// TIA Portal V17 export
// export: Created 2024-09-02T12:50:07.0584181Z, ExportSetting WithDefaults, DisplayName Totally Integrated Automation Portal, DisplayVersion V17, DisplayName TIA Portal Openness, DisplayVersion V17, DisplayName TIA Portal Version Control Interface, DisplayVersion V17, DisplayName STEP 7 Professional, DisplayVersion V17, DisplayName STEP 7 Safety, DisplayVersion V17, DisplayName WinCC Professional, DisplayVersion V17
FUNCTION "AnwFC2_FG01_Station_OP70" : Void   // FC1282, LAD
TITLE = Station
{ S7_Optimized_Access := 'TRUE' }
AUTHOR : VAF
FAMILY : SK
NAME : SK
VERSION : 0.1
// stored: AutoNumber false, IsIECCheckEnabled false, SetENOAutomatically false, UDAEnableTagReadback false
   VAR_TEMP
      Motion_Release : Bool;   // Motion permit
      Hand : Bool;
      Auto : Bool;
      t_Ret_Val_SFC : Int;
      t_fm_Gen : Bool;
      t_ParityFault : Bool;
      t_ConfigFault : Bool;
      t_Retval : Bool;
      MM90_AS : Bool;
      MM90_GS : Bool;
      X1 : Int;
      X2 : Int;
      Y : Int;
      X_actual : Int;
   END_VAR
   VAR_TEMP   // added for the SCL form of the ladder/FBD networks
      _w1 : Bool;
      _w2 : Bool;
   END_VAR
BEGIN

REGION Network 1: Motion permit / Hand/ Auto
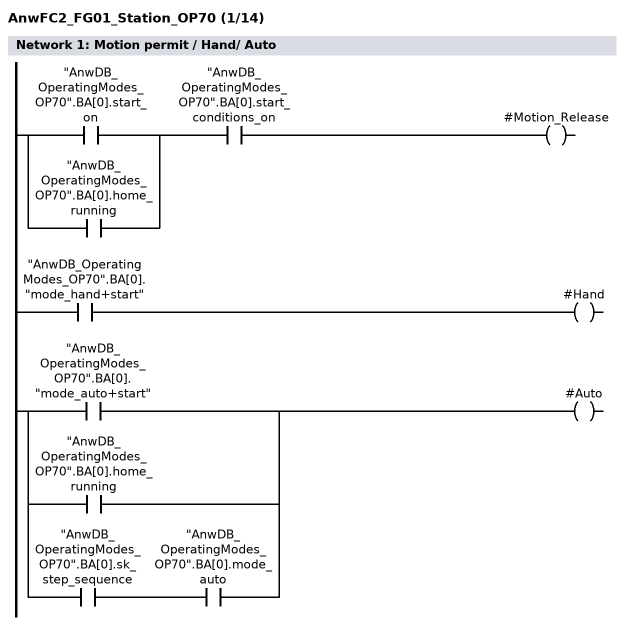
   RUNG wire#powerrail
      Contact( "AnwDB_OperatingModes_OP70".BA[0].start_on )
      wire#w1
      Contact( "AnwDB_OperatingModes_OP70".BA[0].start_conditions_on )
      Coil( #Motion_Release )
   END_RUNG
   RUNG wire#powerrail
      Contact( "AnwDB_OperatingModes_OP70".BA[0].home_running )
   END_RUNG wire#w1
   RUNG wire#powerrail
      Contact( "AnwDB_OperatingModes_OP70".BA[0]."mode_hand+start" )
      Coil( #Hand )
   END_RUNG
   RUNG wire#powerrail
      Contact( "AnwDB_OperatingModes_OP70".BA[0]."mode_auto+start" )
      wire#w2
      Coil( #Auto )
   END_RUNG
   RUNG wire#powerrail
      Contact( "AnwDB_OperatingModes_OP70".BA[0].home_running )
   END_RUNG wire#w2
   RUNG wire#powerrail
      Contact( "AnwDB_OperatingModes_OP70".BA[0].sk_step_sequence )
      Contact( "AnwDB_OperatingModes_OP70".BA[0].mode_auto )
   END_RUNG wire#w2
   // the same network as SCL:
   #Motion_Release := ("AnwDB_OperatingModes_OP70".BA[0].start_on OR "AnwDB_OperatingModes_OP70".BA[0].home_running) AND "AnwDB_OperatingModes_OP70".BA[0].start_conditions_on;
   #Hand := "AnwDB_OperatingModes_OP70".BA[0]."mode_hand+start";
   #Auto := "AnwDB_OperatingModes_OP70".BA[0]."mode_auto+start" OR "AnwDB_OperatingModes_OP70".BA[0].home_running OR ("AnwDB_OperatingModes_OP70".BA[0].sk_step_sequence AND "AnwDB_OperatingModes_OP70".BA[0].mode_auto);
END_REGION

REGION Network 2: Call of the step sequence
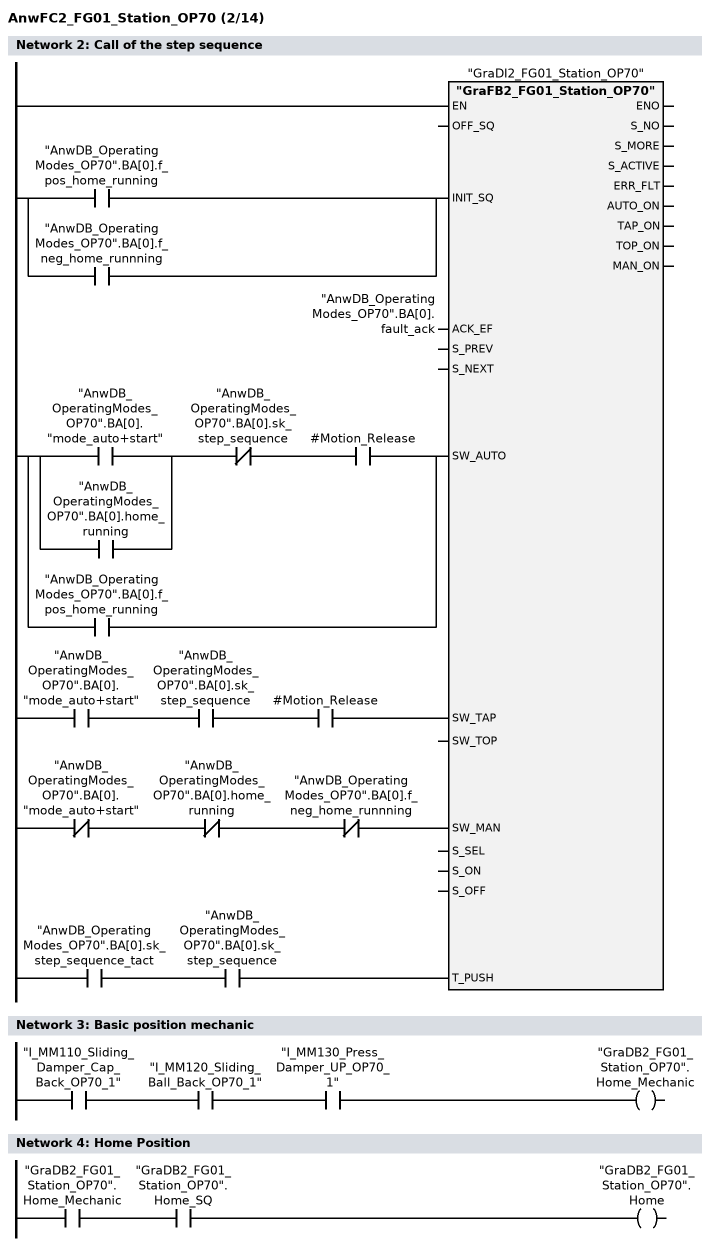
   RUNG wire#powerrail
      "GraDI2_FG01_Station_OP70"(INIT_SQ := wire#w1, SW_AUTO := wire#w3, SW_TAP := wire#w4, SW_MAN := wire#w5, T_PUSH := wire#w6, OFF_SQ :=, ACK_EF := "AnwDB_OperatingModes_OP70".BA[0].fault_ack, S_PREV :=, S_NEXT :=, SW_TOP :=, S_SEL :=, S_ON :=, S_OFF :=, S_NO =>, S_MORE =>, S_ACTIVE =>, ERR_FLT =>, AUTO_ON =>, TAP_ON =>, TOP_ON =>, MAN_ON =>)
   END_RUNG
   RUNG wire#powerrail
      Contact( "AnwDB_OperatingModes_OP70".BA[0].f_pos_home_running )
   END_RUNG wire#w1
   RUNG wire#powerrail
      Contact( "AnwDB_OperatingModes_OP70".BA[0].f_neg_home_runnning )
   END_RUNG wire#w1
   RUNG wire#powerrail
      Contact( "AnwDB_OperatingModes_OP70".BA[0]."mode_auto+start" )
      wire#w2
      I_Contact( "AnwDB_OperatingModes_OP70".BA[0].sk_step_sequence )
      Contact( #Motion_Release )
   END_RUNG wire#w3
   RUNG wire#powerrail
      Contact( "AnwDB_OperatingModes_OP70".BA[0].home_running )
   END_RUNG wire#w2
   RUNG wire#powerrail
      Contact( "AnwDB_OperatingModes_OP70".BA[0].f_pos_home_running )
   END_RUNG wire#w3
   RUNG wire#powerrail
      Contact( "AnwDB_OperatingModes_OP70".BA[0]."mode_auto+start" )
      Contact( "AnwDB_OperatingModes_OP70".BA[0].sk_step_sequence )
      Contact( #Motion_Release )
   END_RUNG wire#w4
   RUNG wire#powerrail
      I_Contact( "AnwDB_OperatingModes_OP70".BA[0]."mode_auto+start" )
      I_Contact( "AnwDB_OperatingModes_OP70".BA[0].home_running )
      I_Contact( "AnwDB_OperatingModes_OP70".BA[0].f_neg_home_runnning )
   END_RUNG wire#w5
   RUNG wire#powerrail
      Contact( "AnwDB_OperatingModes_OP70".BA[0].sk_step_sequence_tact )
      Contact( "AnwDB_OperatingModes_OP70".BA[0].sk_step_sequence )
   END_RUNG wire#w6
   // the same network as SCL:
   "GraDI2_FG01_Station_OP70"(INIT_SQ := "AnwDB_OperatingModes_OP70".BA[0].f_pos_home_running OR "AnwDB_OperatingModes_OP70".BA[0].f_neg_home_runnning,   // "GraFB2_FG01_Station_OP70"
                           ACK_EF := "AnwDB_OperatingModes_OP70".BA[0].fault_ack,
                           SW_AUTO := (("AnwDB_OperatingModes_OP70".BA[0]."mode_auto+start" OR "AnwDB_OperatingModes_OP70".BA[0].home_running) AND NOT "AnwDB_OperatingModes_OP70".BA[0].sk_step_sequence AND #Motion_Release) OR "AnwDB_OperatingModes_OP70".BA[0].f_pos_home_running,
                           SW_TAP := "AnwDB_OperatingModes_OP70".BA[0]."mode_auto+start" AND "AnwDB_OperatingModes_OP70".BA[0].sk_step_sequence AND #Motion_Release,
                           SW_MAN := NOT "AnwDB_OperatingModes_OP70".BA[0]."mode_auto+start" AND NOT "AnwDB_OperatingModes_OP70".BA[0].home_running AND NOT "AnwDB_OperatingModes_OP70".BA[0].f_neg_home_runnning,
                           T_PUSH := "AnwDB_OperatingModes_OP70".BA[0].sk_step_sequence_tact AND "AnwDB_OperatingModes_OP70".BA[0].sk_step_sequence);
END_REGION

REGION Network 3: Basic position mechanic
   RUNG wire#powerrail
      Contact( "I_MM110_Sliding_Damper_Cap_Back_OP70_1" )
      Contact( "I_MM120_Sliding_Ball_Back_OP70_1" )
      Contact( "I_MM130_Press_Damper_UP_OP70_1" )
      Coil( "GraDB2_FG01_Station_OP70".Home_Mechanic )
   END_RUNG
   // the same network as SCL:
   "GraDB2_FG01_Station_OP70".Home_Mechanic := "I_MM110_Sliding_Damper_Cap_Back_OP70_1" AND "I_MM120_Sliding_Ball_Back_OP70_1" AND "I_MM130_Press_Damper_UP_OP70_1";
END_REGION

REGION Network 4: Home Position
   RUNG wire#powerrail
      Contact( "GraDB2_FG01_Station_OP70".Home_Mechanic )
      Contact( "GraDB2_FG01_Station_OP70".Home_SQ )
      Coil( "GraDB2_FG01_Station_OP70".Home )
   END_RUNG
   // the same network as SCL:
   "GraDB2_FG01_Station_OP70".Home := "GraDB2_FG01_Station_OP70".Home_Mechanic AND "GraDB2_FG01_Station_OP70".Home_SQ;
END_REGION

REGION Network 5: ########### USER ###########
END_REGION

REGION Network 6: Screen selection with NOK BEA1
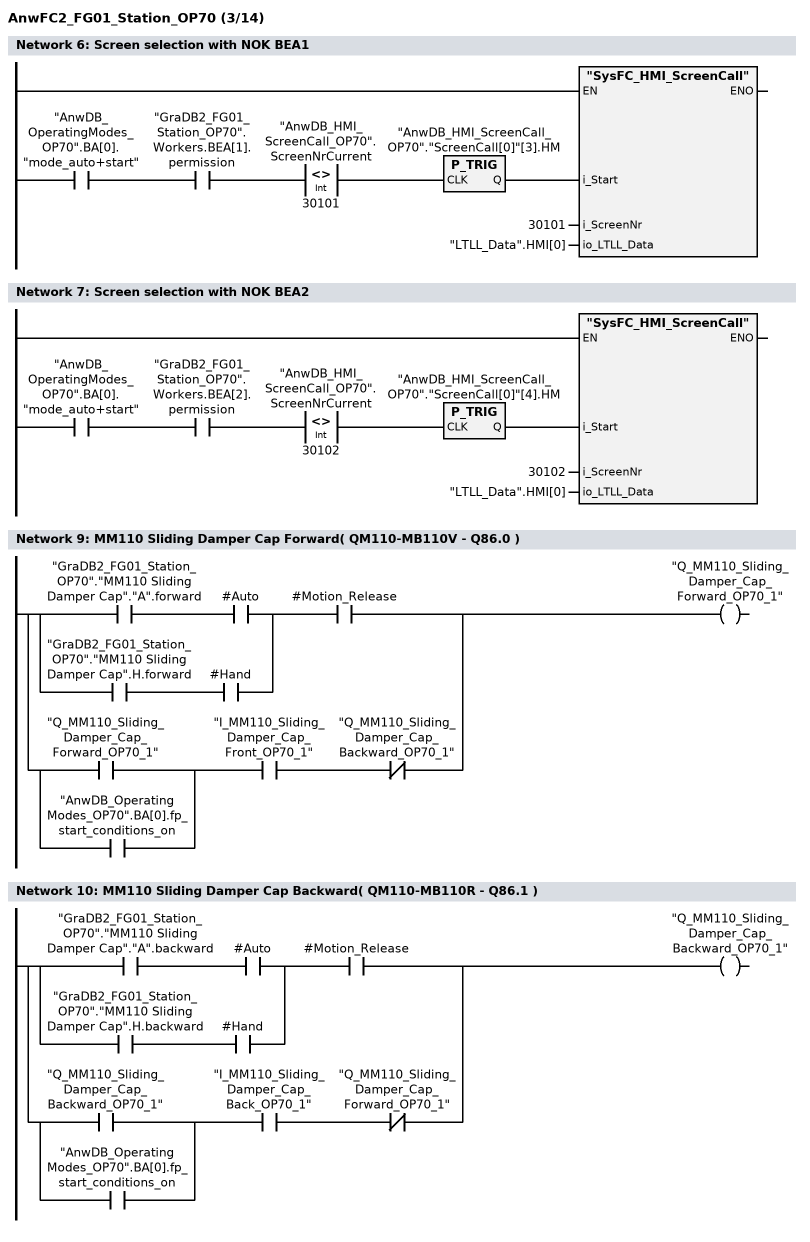
   RUNG wire#powerrail
      "SysFC_HMI_ScreenCall"(i_Start := wire#w1, i_ScreenNr := 30101, io_LTLL_Data := "LTLL_Data".HMI[0])
   END_RUNG
   RUNG wire#powerrail
      Contact( "AnwDB_OperatingModes_OP70".BA[0]."mode_auto+start" )
      Contact( "GraDB2_FG01_Station_OP70".Workers.BEA[1].permission )
      { S7_Templates := "SrcType := Int" } NE_Contact(in1 := "AnwDB_HMI_ScreenCall_OP70".ScreenNrCurrent, in2 := 30101)
      P_Trig( "AnwDB_HMI_ScreenCall_OP70"."ScreenCall[0]"[3].HM )
   END_RUNG wire#w1
   // the same network as SCL:
   #_w1 := "AnwDB_OperatingModes_OP70".BA[0]."mode_auto+start" AND "GraDB2_FG01_Station_OP70".Workers.BEA[1].permission AND ("AnwDB_HMI_ScreenCall_OP70".ScreenNrCurrent <> 30101);
   #_w2 := #_w1 AND NOT "AnwDB_HMI_ScreenCall_OP70"."ScreenCall[0]"[3].HM;   // rising edge
   "AnwDB_HMI_ScreenCall_OP70"."ScreenCall[0]"[3].HM := #_w1;
   "SysFC_HMI_ScreenCall"(i_Start := #_w2, i_ScreenNr := 30101, io_LTLL_Data := "LTLL_Data".HMI[0]);
END_REGION

REGION Network 7: Screen selection with NOK BEA2
   RUNG wire#powerrail
      "SysFC_HMI_ScreenCall"(i_Start := wire#w1, i_ScreenNr := 30102, io_LTLL_Data := "LTLL_Data".HMI[0])
   END_RUNG
   RUNG wire#powerrail
      Contact( "AnwDB_OperatingModes_OP70".BA[0]."mode_auto+start" )
      Contact( "GraDB2_FG01_Station_OP70".Workers.BEA[2].permission )
      { S7_Templates := "SrcType := Int" } NE_Contact(in1 := "AnwDB_HMI_ScreenCall_OP70".ScreenNrCurrent, in2 := 30102)
      P_Trig( "AnwDB_HMI_ScreenCall_OP70"."ScreenCall[0]"[4].HM )
   END_RUNG wire#w1
   // the same network as SCL:
   #_w1 := "AnwDB_OperatingModes_OP70".BA[0]."mode_auto+start" AND "GraDB2_FG01_Station_OP70".Workers.BEA[2].permission AND ("AnwDB_HMI_ScreenCall_OP70".ScreenNrCurrent <> 30102);
   #_w2 := #_w1 AND NOT "AnwDB_HMI_ScreenCall_OP70"."ScreenCall[0]"[4].HM;   // rising edge
   "AnwDB_HMI_ScreenCall_OP70"."ScreenCall[0]"[4].HM := #_w1;
   "SysFC_HMI_ScreenCall"(i_Start := #_w2, i_ScreenNr := 30102, io_LTLL_Data := "LTLL_Data".HMI[0]);
END_REGION

REGION Network 8: ########### SS_02_001_Setup ###########
END_REGION

REGION Network 9: MM110 Sliding Damper Cap Forward( QM110-MB110V - Q86.0 )
   RUNG wire#powerrail
      Contact( "GraDB2_FG01_Station_OP70"."MM110 Sliding Damper Cap"."A".forward )
      Contact( #Auto )
      wire#w1
      Contact( #Motion_Release )
      wire#w2
      Coil( "Q_MM110_Sliding_Damper_Cap_Forward_OP70_1" )
   END_RUNG
   RUNG wire#powerrail
      Contact( "GraDB2_FG01_Station_OP70"."MM110 Sliding Damper Cap".H.forward )
      Contact( #Hand )
   END_RUNG wire#w1
   RUNG wire#powerrail
      Contact( "Q_MM110_Sliding_Damper_Cap_Forward_OP70_1" )
      wire#w3
      Contact( "I_MM110_Sliding_Damper_Cap_Front_OP70_1" )
      I_Contact( "Q_MM110_Sliding_Damper_Cap_Backward_OP70_1" )
   END_RUNG wire#w2
   RUNG wire#powerrail
      Contact( "AnwDB_OperatingModes_OP70".BA[0].fp_start_conditions_on )
   END_RUNG wire#w3
   // the same network as SCL:
   "Q_MM110_Sliding_Damper_Cap_Forward_OP70_1" := ((("GraDB2_FG01_Station_OP70"."MM110 Sliding Damper Cap"."A".forward AND #Auto) OR ("GraDB2_FG01_Station_OP70"."MM110 Sliding Damper Cap".H.forward AND #Hand)) AND #Motion_Release) OR (("Q_MM110_Sliding_Damper_Cap_Forward_OP70_1" OR "AnwDB_OperatingModes_OP70".BA[0].fp_start_conditions_on) AND "I_MM110_Sliding_Damper_Cap_Front_OP70_1" AND NOT "Q_MM110_Sliding_Damper_Cap_Backward_OP70_1");
END_REGION

REGION Network 10: MM110 Sliding Damper Cap Backward( QM110-MB110R - Q86.1 )
   RUNG wire#powerrail
      Contact( "GraDB2_FG01_Station_OP70"."MM110 Sliding Damper Cap"."A".backward )
      Contact( #Auto )
      wire#w1
      Contact( #Motion_Release )
      wire#w2
      Coil( "Q_MM110_Sliding_Damper_Cap_Backward_OP70_1" )
   END_RUNG
   RUNG wire#powerrail
      Contact( "GraDB2_FG01_Station_OP70"."MM110 Sliding Damper Cap".H.backward )
      Contact( #Hand )
   END_RUNG wire#w1
   RUNG wire#powerrail
      Contact( "Q_MM110_Sliding_Damper_Cap_Backward_OP70_1" )
      wire#w3
      Contact( "I_MM110_Sliding_Damper_Cap_Back_OP70_1" )
      I_Contact( "Q_MM110_Sliding_Damper_Cap_Forward_OP70_1" )
   END_RUNG wire#w2
   RUNG wire#powerrail
      Contact( "AnwDB_OperatingModes_OP70".BA[0].fp_start_conditions_on )
   END_RUNG wire#w3
   // the same network as SCL:
   "Q_MM110_Sliding_Damper_Cap_Backward_OP70_1" := ((("GraDB2_FG01_Station_OP70"."MM110 Sliding Damper Cap"."A".backward AND #Auto) OR ("GraDB2_FG01_Station_OP70"."MM110 Sliding Damper Cap".H.backward AND #Hand)) AND #Motion_Release) OR (("Q_MM110_Sliding_Damper_Cap_Backward_OP70_1" OR "AnwDB_OperatingModes_OP70".BA[0].fp_start_conditions_on) AND "I_MM110_Sliding_Damper_Cap_Back_OP70_1" AND NOT "Q_MM110_Sliding_Damper_Cap_Forward_OP70_1");
END_REGION

REGION Network 11: Hand line(13)
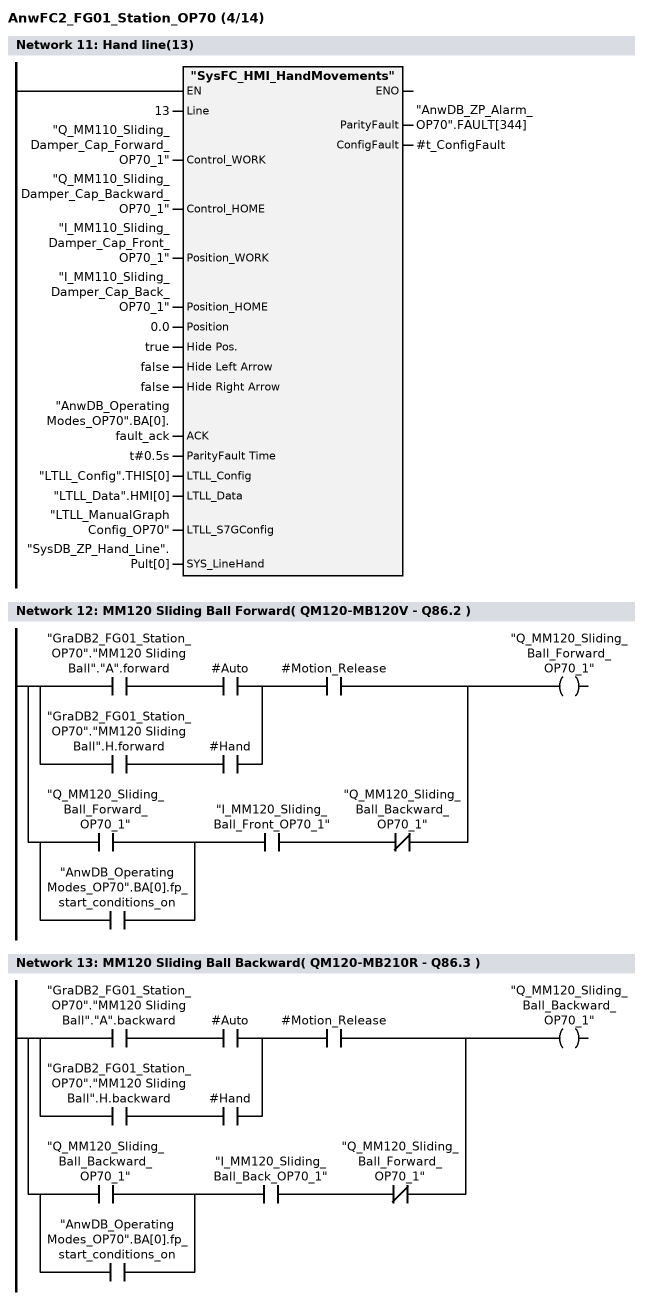
   RUNG wire#powerrail
      "SysFC_HMI_HandMovements"(Line := 13, Control_WORK := "Q_MM110_Sliding_Damper_Cap_Forward_OP70_1", Control_HOME := "Q_MM110_Sliding_Damper_Cap_Backward_OP70_1", Position_WORK := "I_MM110_Sliding_Damper_Cap_Front_OP70_1", Position_HOME := "I_MM110_Sliding_Damper_Cap_Back_OP70_1", Position := 0.0, "Hide Pos." := true, "Hide Left Arrow" := false, "Hide Right Arrow" := false, ACK := "AnwDB_OperatingModes_OP70".BA[0].fault_ack, "ParityFault Time" := t#0.5s, LTLL_Config := "LTLL_Config".THIS[0], LTLL_Data := "LTLL_Data".HMI[0], LTLL_S7GConfig := "LTLL_ManualGraphConfig_OP70", SYS_LineHand := "SysDB_ZP_Hand_Line".Pult[0], ParityFault => "AnwDB_ZP_Alarm_OP70".FAULT[344], ConfigFault => #t_ConfigFault)
   END_RUNG
   // the same network as SCL:
   "SysFC_HMI_HandMovements"(Line := 13,
                           Control_WORK := "Q_MM110_Sliding_Damper_Cap_Forward_OP70_1",
                           Control_HOME := "Q_MM110_Sliding_Damper_Cap_Backward_OP70_1",
                           Position_WORK := "I_MM110_Sliding_Damper_Cap_Front_OP70_1",
                           Position_HOME := "I_MM110_Sliding_Damper_Cap_Back_OP70_1",
                           Position := 0.0,
                           "Hide Pos." := true,
                           "Hide Left Arrow" := false,
                           "Hide Right Arrow" := false,
                           ACK := "AnwDB_OperatingModes_OP70".BA[0].fault_ack,
                           "ParityFault Time" := t#0.5s,
                           LTLL_Config := "LTLL_Config".THIS[0],
                           LTLL_Data := "LTLL_Data".HMI[0],
                           LTLL_S7GConfig := "LTLL_ManualGraphConfig_OP70",
                           SYS_LineHand := "SysDB_ZP_Hand_Line".Pult[0],
                           ParityFault => "AnwDB_ZP_Alarm_OP70".FAULT[344],
                           ConfigFault => #t_ConfigFault);
END_REGION

REGION Network 12: MM120 Sliding Ball Forward( QM120-MB120V - Q86.2 )
   RUNG wire#powerrail
      Contact( "GraDB2_FG01_Station_OP70"."MM120 Sliding Ball"."A".forward )
      Contact( #Auto )
      wire#w1
      Contact( #Motion_Release )
      wire#w2
      Coil( "Q_MM120_Sliding_Ball_Forward_OP70_1" )
   END_RUNG
   RUNG wire#powerrail
      Contact( "GraDB2_FG01_Station_OP70"."MM120 Sliding Ball".H.forward )
      Contact( #Hand )
   END_RUNG wire#w1
   RUNG wire#powerrail
      Contact( "Q_MM120_Sliding_Ball_Forward_OP70_1" )
      wire#w3
      Contact( "I_MM120_Sliding_Ball_Front_OP70_1" )
      I_Contact( "Q_MM120_Sliding_Ball_Backward_OP70_1" )
   END_RUNG wire#w2
   RUNG wire#powerrail
      Contact( "AnwDB_OperatingModes_OP70".BA[0].fp_start_conditions_on )
   END_RUNG wire#w3
   // the same network as SCL:
   "Q_MM120_Sliding_Ball_Forward_OP70_1" := ((("GraDB2_FG01_Station_OP70"."MM120 Sliding Ball"."A".forward AND #Auto) OR ("GraDB2_FG01_Station_OP70"."MM120 Sliding Ball".H.forward AND #Hand)) AND #Motion_Release) OR (("Q_MM120_Sliding_Ball_Forward_OP70_1" OR "AnwDB_OperatingModes_OP70".BA[0].fp_start_conditions_on) AND "I_MM120_Sliding_Ball_Front_OP70_1" AND NOT "Q_MM120_Sliding_Ball_Backward_OP70_1");
END_REGION

REGION Network 13: MM120 Sliding Ball Backward( QM120-MB210R - Q86.3 )
   RUNG wire#powerrail
      Contact( "GraDB2_FG01_Station_OP70"."MM120 Sliding Ball"."A".backward )
      Contact( #Auto )
      wire#w1
      Contact( #Motion_Release )
      wire#w2
      Coil( "Q_MM120_Sliding_Ball_Backward_OP70_1" )
   END_RUNG
   RUNG wire#powerrail
      Contact( "GraDB2_FG01_Station_OP70"."MM120 Sliding Ball".H.backward )
      Contact( #Hand )
   END_RUNG wire#w1
   RUNG wire#powerrail
      Contact( "Q_MM120_Sliding_Ball_Backward_OP70_1" )
      wire#w3
      Contact( "I_MM120_Sliding_Ball_Back_OP70_1" )
      I_Contact( "Q_MM120_Sliding_Ball_Forward_OP70_1" )
   END_RUNG wire#w2
   RUNG wire#powerrail
      Contact( "AnwDB_OperatingModes_OP70".BA[0].fp_start_conditions_on )
   END_RUNG wire#w3
   // the same network as SCL:
   "Q_MM120_Sliding_Ball_Backward_OP70_1" := ((("GraDB2_FG01_Station_OP70"."MM120 Sliding Ball"."A".backward AND #Auto) OR ("GraDB2_FG01_Station_OP70"."MM120 Sliding Ball".H.backward AND #Hand)) AND #Motion_Release) OR (("Q_MM120_Sliding_Ball_Backward_OP70_1" OR "AnwDB_OperatingModes_OP70".BA[0].fp_start_conditions_on) AND "I_MM120_Sliding_Ball_Back_OP70_1" AND NOT "Q_MM120_Sliding_Ball_Forward_OP70_1");
END_REGION

REGION Network 14: Hand line(14)
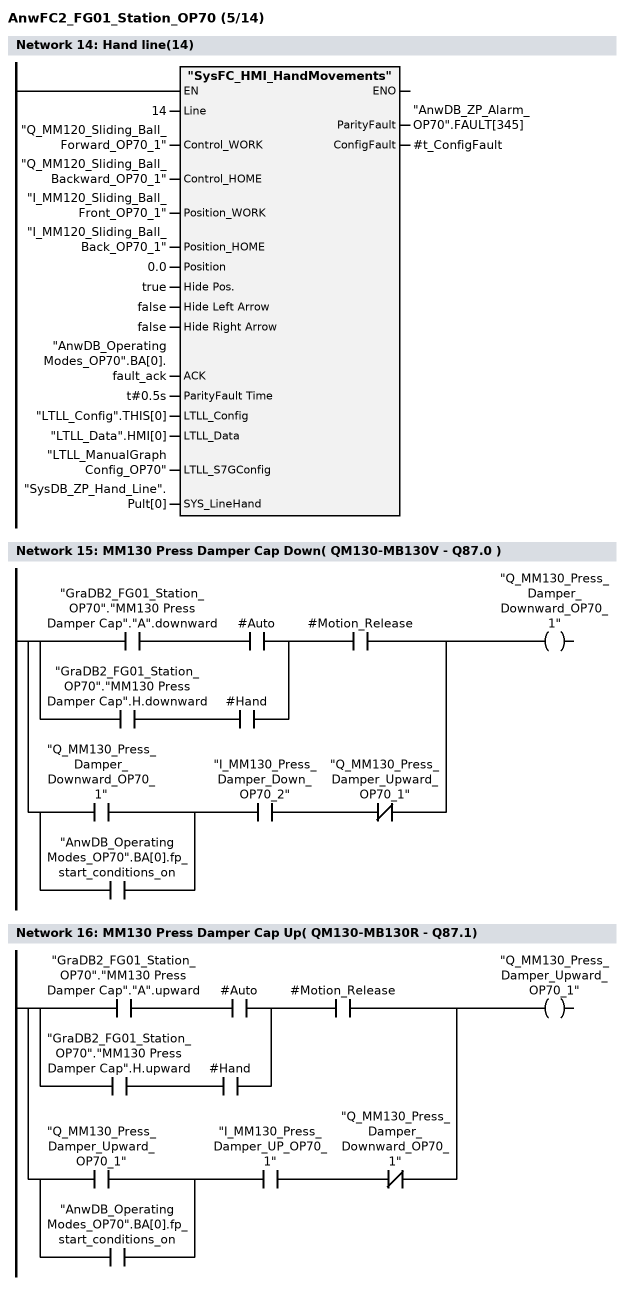
   RUNG wire#powerrail
      "SysFC_HMI_HandMovements"(Line := 14, Control_WORK := "Q_MM120_Sliding_Ball_Forward_OP70_1", Control_HOME := "Q_MM120_Sliding_Ball_Backward_OP70_1", Position_WORK := "I_MM120_Sliding_Ball_Front_OP70_1", Position_HOME := "I_MM120_Sliding_Ball_Back_OP70_1", Position := 0.0, "Hide Pos." := true, "Hide Left Arrow" := false, "Hide Right Arrow" := false, ACK := "AnwDB_OperatingModes_OP70".BA[0].fault_ack, "ParityFault Time" := t#0.5s, LTLL_Config := "LTLL_Config".THIS[0], LTLL_Data := "LTLL_Data".HMI[0], LTLL_S7GConfig := "LTLL_ManualGraphConfig_OP70", SYS_LineHand := "SysDB_ZP_Hand_Line".Pult[0], ParityFault => "AnwDB_ZP_Alarm_OP70".FAULT[345], ConfigFault => #t_ConfigFault)
   END_RUNG
   // the same network as SCL:
   "SysFC_HMI_HandMovements"(Line := 14,
                           Control_WORK := "Q_MM120_Sliding_Ball_Forward_OP70_1",
                           Control_HOME := "Q_MM120_Sliding_Ball_Backward_OP70_1",
                           Position_WORK := "I_MM120_Sliding_Ball_Front_OP70_1",
                           Position_HOME := "I_MM120_Sliding_Ball_Back_OP70_1",
                           Position := 0.0,
                           "Hide Pos." := true,
                           "Hide Left Arrow" := false,
                           "Hide Right Arrow" := false,
                           ACK := "AnwDB_OperatingModes_OP70".BA[0].fault_ack,
                           "ParityFault Time" := t#0.5s,
                           LTLL_Config := "LTLL_Config".THIS[0],
                           LTLL_Data := "LTLL_Data".HMI[0],
                           LTLL_S7GConfig := "LTLL_ManualGraphConfig_OP70",
                           SYS_LineHand := "SysDB_ZP_Hand_Line".Pult[0],
                           ParityFault => "AnwDB_ZP_Alarm_OP70".FAULT[345],
                           ConfigFault => #t_ConfigFault);
END_REGION

REGION Network 15: MM130 Press Damper Cap Down( QM130-MB130V - Q87.0 )
   RUNG wire#powerrail
      Contact( "GraDB2_FG01_Station_OP70"."MM130 Press Damper Cap"."A".downward )
      Contact( #Auto )
      wire#w1
      Contact( #Motion_Release )
      wire#w2
      Coil( "Q_MM130_Press_Damper_Downward_OP70_1" )
   END_RUNG
   RUNG wire#powerrail
      Contact( "GraDB2_FG01_Station_OP70"."MM130 Press Damper Cap".H.downward )
      Contact( #Hand )
   END_RUNG wire#w1
   RUNG wire#powerrail
      Contact( "Q_MM130_Press_Damper_Downward_OP70_1" )
      wire#w3
      Contact( "I_MM130_Press_Damper_Down_OP70_2" )
      I_Contact( "Q_MM130_Press_Damper_Upward_OP70_1" )
   END_RUNG wire#w2
   RUNG wire#powerrail
      Contact( "AnwDB_OperatingModes_OP70".BA[0].fp_start_conditions_on )
   END_RUNG wire#w3
   // the same network as SCL:
   "Q_MM130_Press_Damper_Downward_OP70_1" := ((("GraDB2_FG01_Station_OP70"."MM130 Press Damper Cap"."A".downward AND #Auto) OR ("GraDB2_FG01_Station_OP70"."MM130 Press Damper Cap".H.downward AND #Hand)) AND #Motion_Release) OR (("Q_MM130_Press_Damper_Downward_OP70_1" OR "AnwDB_OperatingModes_OP70".BA[0].fp_start_conditions_on) AND "I_MM130_Press_Damper_Down_OP70_2" AND NOT "Q_MM130_Press_Damper_Upward_OP70_1");
END_REGION

REGION Network 16: MM130 Press Damper Cap Up( QM130-MB130R - Q87.1)
   RUNG wire#powerrail
      Contact( "GraDB2_FG01_Station_OP70"."MM130 Press Damper Cap"."A".upward )
      Contact( #Auto )
      wire#w1
      Contact( #Motion_Release )
      wire#w2
      Coil( "Q_MM130_Press_Damper_Upward_OP70_1" )
   END_RUNG
   RUNG wire#powerrail
      Contact( "GraDB2_FG01_Station_OP70"."MM130 Press Damper Cap".H.upward )
      Contact( #Hand )
   END_RUNG wire#w1
   RUNG wire#powerrail
      Contact( "Q_MM130_Press_Damper_Upward_OP70_1" )
      wire#w3
      Contact( "I_MM130_Press_Damper_UP_OP70_1" )
      I_Contact( "Q_MM130_Press_Damper_Downward_OP70_1" )
   END_RUNG wire#w2
   RUNG wire#powerrail
      Contact( "AnwDB_OperatingModes_OP70".BA[0].fp_start_conditions_on )
   END_RUNG wire#w3
   // the same network as SCL:
   "Q_MM130_Press_Damper_Upward_OP70_1" := ((("GraDB2_FG01_Station_OP70"."MM130 Press Damper Cap"."A".upward AND #Auto) OR ("GraDB2_FG01_Station_OP70"."MM130 Press Damper Cap".H.upward AND #Hand)) AND #Motion_Release) OR (("Q_MM130_Press_Damper_Upward_OP70_1" OR "AnwDB_OperatingModes_OP70".BA[0].fp_start_conditions_on) AND "I_MM130_Press_Damper_UP_OP70_1" AND NOT "Q_MM130_Press_Damper_Downward_OP70_1");
END_REGION

REGION Network 17: Hand line(15)
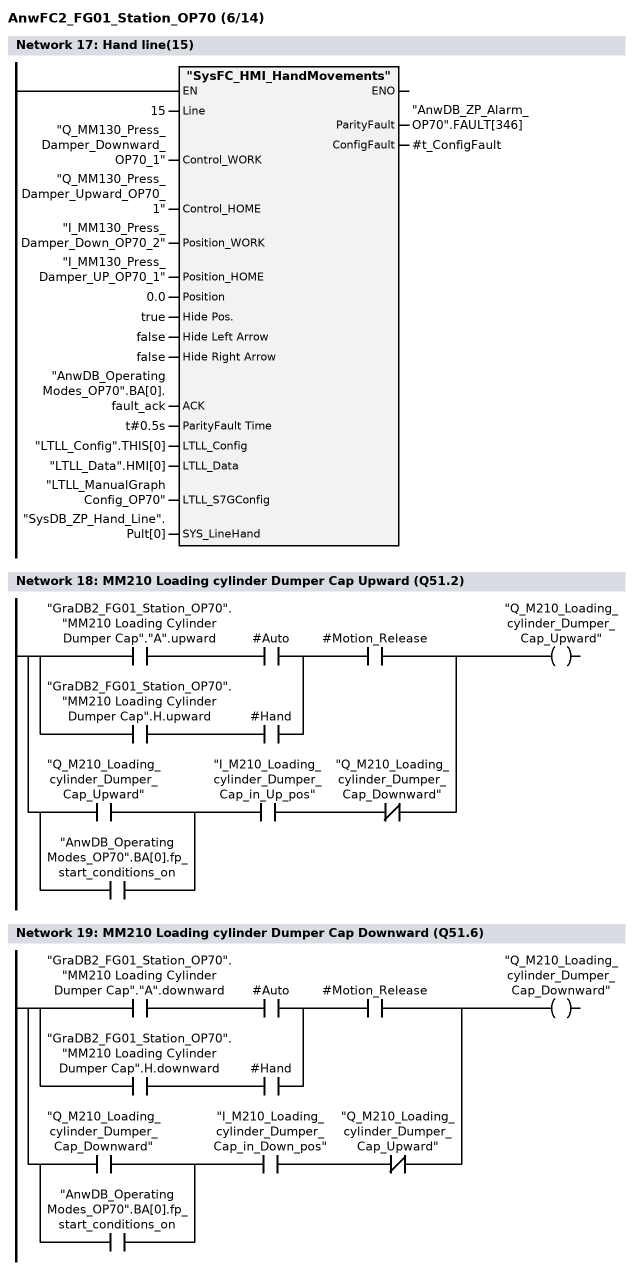
   RUNG wire#powerrail
      "SysFC_HMI_HandMovements"(Line := 15, Control_WORK := "Q_MM130_Press_Damper_Downward_OP70_1", Control_HOME := "Q_MM130_Press_Damper_Upward_OP70_1", Position_WORK := "I_MM130_Press_Damper_Down_OP70_2", Position_HOME := "I_MM130_Press_Damper_UP_OP70_1", Position := 0.0, "Hide Pos." := true, "Hide Left Arrow" := false, "Hide Right Arrow" := false, ACK := "AnwDB_OperatingModes_OP70".BA[0].fault_ack, "ParityFault Time" := t#0.5s, LTLL_Config := "LTLL_Config".THIS[0], LTLL_Data := "LTLL_Data".HMI[0], LTLL_S7GConfig := "LTLL_ManualGraphConfig_OP70", SYS_LineHand := "SysDB_ZP_Hand_Line".Pult[0], ParityFault => "AnwDB_ZP_Alarm_OP70".FAULT[346], ConfigFault => #t_ConfigFault)
   END_RUNG
   // the same network as SCL:
   "SysFC_HMI_HandMovements"(Line := 15,
                           Control_WORK := "Q_MM130_Press_Damper_Downward_OP70_1",
                           Control_HOME := "Q_MM130_Press_Damper_Upward_OP70_1",
                           Position_WORK := "I_MM130_Press_Damper_Down_OP70_2",
                           Position_HOME := "I_MM130_Press_Damper_UP_OP70_1",
                           Position := 0.0,
                           "Hide Pos." := true,
                           "Hide Left Arrow" := false,
                           "Hide Right Arrow" := false,
                           ACK := "AnwDB_OperatingModes_OP70".BA[0].fault_ack,
                           "ParityFault Time" := t#0.5s,
                           LTLL_Config := "LTLL_Config".THIS[0],
                           LTLL_Data := "LTLL_Data".HMI[0],
                           LTLL_S7GConfig := "LTLL_ManualGraphConfig_OP70",
                           SYS_LineHand := "SysDB_ZP_Hand_Line".Pult[0],
                           ParityFault => "AnwDB_ZP_Alarm_OP70".FAULT[346],
                           ConfigFault => #t_ConfigFault);
END_REGION

REGION Network 18: MM210 Loading cylinder Dumper Cap Upward (Q51.2)
   RUNG wire#powerrail
      Contact( "GraDB2_FG01_Station_OP70"."MM210 Loading Cylinder Dumper Cap"."A".upward )
      Contact( #Auto )
      wire#w1
      Contact( #Motion_Release )
      wire#w2
      Coil( "Q_M210_Loading_cylinder_Dumper_Cap_Upward" )
   END_RUNG
   RUNG wire#powerrail
      Contact( "GraDB2_FG01_Station_OP70"."MM210 Loading Cylinder Dumper Cap".H.upward )
      Contact( #Hand )
   END_RUNG wire#w1
   RUNG wire#powerrail
      Contact( "Q_M210_Loading_cylinder_Dumper_Cap_Upward" )
      wire#w3
      Contact( "I_M210_Loading_cylinder_Dumper_Cap_in_Up_pos" )
      I_Contact( "Q_M210_Loading_cylinder_Dumper_Cap_Downward" )
   END_RUNG wire#w2
   RUNG wire#powerrail
      Contact( "AnwDB_OperatingModes_OP70".BA[0].fp_start_conditions_on )
   END_RUNG wire#w3
   // the same network as SCL:
   "Q_M210_Loading_cylinder_Dumper_Cap_Upward" := ((("GraDB2_FG01_Station_OP70"."MM210 Loading Cylinder Dumper Cap"."A".upward AND #Auto) OR ("GraDB2_FG01_Station_OP70"."MM210 Loading Cylinder Dumper Cap".H.upward AND #Hand)) AND #Motion_Release) OR (("Q_M210_Loading_cylinder_Dumper_Cap_Upward" OR "AnwDB_OperatingModes_OP70".BA[0].fp_start_conditions_on) AND "I_M210_Loading_cylinder_Dumper_Cap_in_Up_pos" AND NOT "Q_M210_Loading_cylinder_Dumper_Cap_Downward");
END_REGION

REGION Network 19: MM210 Loading cylinder Dumper Cap Downward (Q51.6)
   RUNG wire#powerrail
      Contact( "GraDB2_FG01_Station_OP70"."MM210 Loading Cylinder Dumper Cap"."A".downward )
      Contact( #Auto )
      wire#w1
      Contact( #Motion_Release )
      wire#w2
      Coil( "Q_M210_Loading_cylinder_Dumper_Cap_Downward" )
   END_RUNG
   RUNG wire#powerrail
      Contact( "GraDB2_FG01_Station_OP70"."MM210 Loading Cylinder Dumper Cap".H.downward )
      Contact( #Hand )
   END_RUNG wire#w1
   RUNG wire#powerrail
      Contact( "Q_M210_Loading_cylinder_Dumper_Cap_Downward" )
      wire#w3
      Contact( "I_M210_Loading_cylinder_Dumper_Cap_in_Down_pos" )
      I_Contact( "Q_M210_Loading_cylinder_Dumper_Cap_Upward" )
   END_RUNG wire#w2
   RUNG wire#powerrail
      Contact( "AnwDB_OperatingModes_OP70".BA[0].fp_start_conditions_on )
   END_RUNG wire#w3
   // the same network as SCL:
   "Q_M210_Loading_cylinder_Dumper_Cap_Downward" := ((("GraDB2_FG01_Station_OP70"."MM210 Loading Cylinder Dumper Cap"."A".downward AND #Auto) OR ("GraDB2_FG01_Station_OP70"."MM210 Loading Cylinder Dumper Cap".H.downward AND #Hand)) AND #Motion_Release) OR (("Q_M210_Loading_cylinder_Dumper_Cap_Downward" OR "AnwDB_OperatingModes_OP70".BA[0].fp_start_conditions_on) AND "I_M210_Loading_cylinder_Dumper_Cap_in_Down_pos" AND NOT "Q_M210_Loading_cylinder_Dumper_Cap_Upward");
END_REGION

REGION Network 20: Hand linie (16)
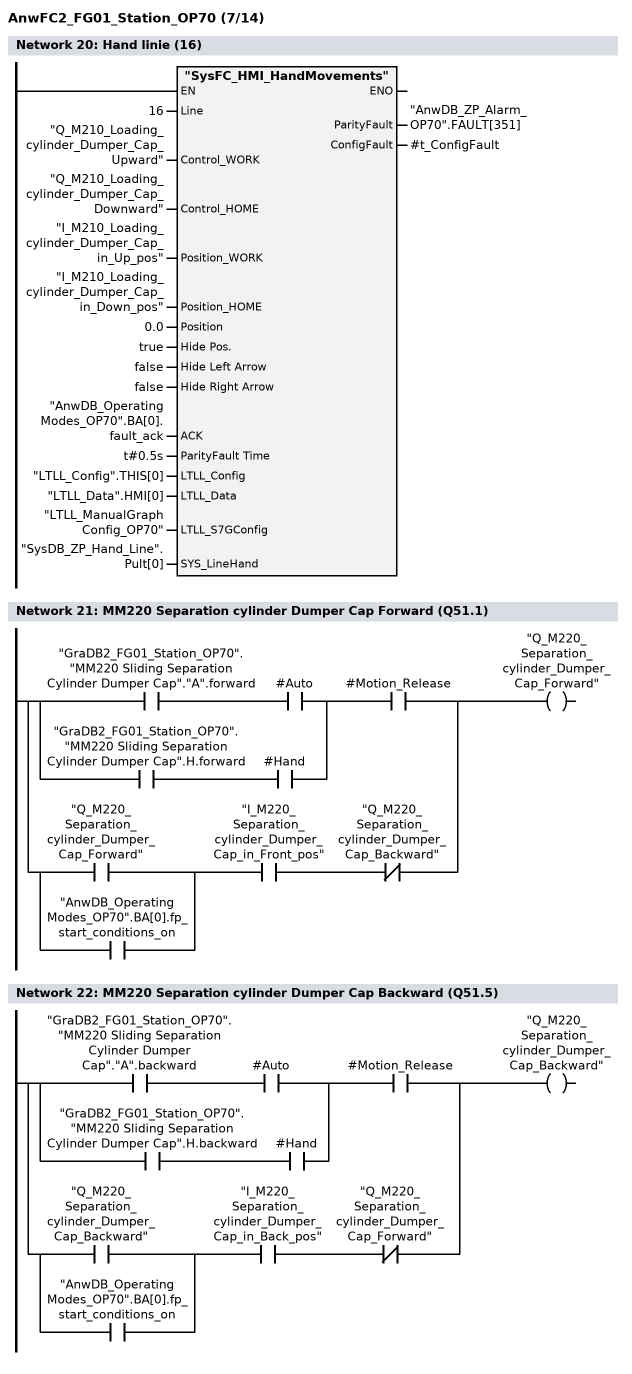
   RUNG wire#powerrail
      "SysFC_HMI_HandMovements"(Line := 16, Control_WORK := "Q_M210_Loading_cylinder_Dumper_Cap_Upward", Control_HOME := "Q_M210_Loading_cylinder_Dumper_Cap_Downward", Position_WORK := "I_M210_Loading_cylinder_Dumper_Cap_in_Up_pos", Position_HOME := "I_M210_Loading_cylinder_Dumper_Cap_in_Down_pos", Position := 0.0, "Hide Pos." := true, "Hide Left Arrow" := false, "Hide Right Arrow" := false, ACK := "AnwDB_OperatingModes_OP70".BA[0].fault_ack, "ParityFault Time" := t#0.5s, LTLL_Config := "LTLL_Config".THIS[0], LTLL_Data := "LTLL_Data".HMI[0], LTLL_S7GConfig := "LTLL_ManualGraphConfig_OP70", SYS_LineHand := "SysDB_ZP_Hand_Line".Pult[0], ParityFault => "AnwDB_ZP_Alarm_OP70".FAULT[351], ConfigFault => #t_ConfigFault)
   END_RUNG
   // the same network as SCL:
   "SysFC_HMI_HandMovements"(Line := 16,
                           Control_WORK := "Q_M210_Loading_cylinder_Dumper_Cap_Upward",
                           Control_HOME := "Q_M210_Loading_cylinder_Dumper_Cap_Downward",
                           Position_WORK := "I_M210_Loading_cylinder_Dumper_Cap_in_Up_pos",
                           Position_HOME := "I_M210_Loading_cylinder_Dumper_Cap_in_Down_pos",
                           Position := 0.0,
                           "Hide Pos." := true,
                           "Hide Left Arrow" := false,
                           "Hide Right Arrow" := false,
                           ACK := "AnwDB_OperatingModes_OP70".BA[0].fault_ack,
                           "ParityFault Time" := t#0.5s,
                           LTLL_Config := "LTLL_Config".THIS[0],
                           LTLL_Data := "LTLL_Data".HMI[0],
                           LTLL_S7GConfig := "LTLL_ManualGraphConfig_OP70",
                           SYS_LineHand := "SysDB_ZP_Hand_Line".Pult[0],
                           ParityFault => "AnwDB_ZP_Alarm_OP70".FAULT[351],
                           ConfigFault => #t_ConfigFault);
END_REGION

REGION Network 21: MM220 Separation cylinder Dumper Cap Forward (Q51.1)
   RUNG wire#powerrail
      Contact( "GraDB2_FG01_Station_OP70"."MM220 Sliding Separation Cylinder Dumper Cap"."A".forward )
      Contact( #Auto )
      wire#w1
      Contact( #Motion_Release )
      wire#w2
      Coil( "Q_M220_Separation_cylinder_Dumper_Cap_Forward" )
   END_RUNG
   RUNG wire#powerrail
      Contact( "GraDB2_FG01_Station_OP70"."MM220 Sliding Separation Cylinder Dumper Cap".H.forward )
      Contact( #Hand )
   END_RUNG wire#w1
   RUNG wire#powerrail
      Contact( "Q_M220_Separation_cylinder_Dumper_Cap_Forward" )
      wire#w3
      Contact( "I_M220_Separation_cylinder_Dumper_Cap_in_Front_pos" )
      I_Contact( "Q_M220_Separation_cylinder_Dumper_Cap_Backward" )
   END_RUNG wire#w2
   RUNG wire#powerrail
      Contact( "AnwDB_OperatingModes_OP70".BA[0].fp_start_conditions_on )
   END_RUNG wire#w3
   // the same network as SCL:
   "Q_M220_Separation_cylinder_Dumper_Cap_Forward" := ((("GraDB2_FG01_Station_OP70"."MM220 Sliding Separation Cylinder Dumper Cap"."A".forward AND #Auto) OR ("GraDB2_FG01_Station_OP70"."MM220 Sliding Separation Cylinder Dumper Cap".H.forward AND #Hand)) AND #Motion_Release) OR (("Q_M220_Separation_cylinder_Dumper_Cap_Forward" OR "AnwDB_OperatingModes_OP70".BA[0].fp_start_conditions_on) AND "I_M220_Separation_cylinder_Dumper_Cap_in_Front_pos" AND NOT "Q_M220_Separation_cylinder_Dumper_Cap_Backward");
END_REGION

REGION Network 22: MM220 Separation cylinder Dumper Cap Backward (Q51.5)
   RUNG wire#powerrail
      Contact( "GraDB2_FG01_Station_OP70"."MM220 Sliding Separation Cylinder Dumper Cap"."A".backward )
      Contact( #Auto )
      wire#w1
      Contact( #Motion_Release )
      wire#w2
      Coil( "Q_M220_Separation_cylinder_Dumper_Cap_Backward" )
   END_RUNG
   RUNG wire#powerrail
      Contact( "GraDB2_FG01_Station_OP70"."MM220 Sliding Separation Cylinder Dumper Cap".H.backward )
      Contact( #Hand )
   END_RUNG wire#w1
   RUNG wire#powerrail
      Contact( "Q_M220_Separation_cylinder_Dumper_Cap_Backward" )
      wire#w3
      Contact( "I_M220_Separation_cylinder_Dumper_Cap_in_Back_pos" )
      I_Contact( "Q_M220_Separation_cylinder_Dumper_Cap_Forward" )
   END_RUNG wire#w2
   RUNG wire#powerrail
      Contact( "AnwDB_OperatingModes_OP70".BA[0].fp_start_conditions_on )
   END_RUNG wire#w3
   // the same network as SCL:
   "Q_M220_Separation_cylinder_Dumper_Cap_Backward" := ((("GraDB2_FG01_Station_OP70"."MM220 Sliding Separation Cylinder Dumper Cap"."A".backward AND #Auto) OR ("GraDB2_FG01_Station_OP70"."MM220 Sliding Separation Cylinder Dumper Cap".H.backward AND #Hand)) AND #Motion_Release) OR (("Q_M220_Separation_cylinder_Dumper_Cap_Backward" OR "AnwDB_OperatingModes_OP70".BA[0].fp_start_conditions_on) AND "I_M220_Separation_cylinder_Dumper_Cap_in_Back_pos" AND NOT "Q_M220_Separation_cylinder_Dumper_Cap_Forward");
END_REGION

REGION Network 23: Hand linie (17)
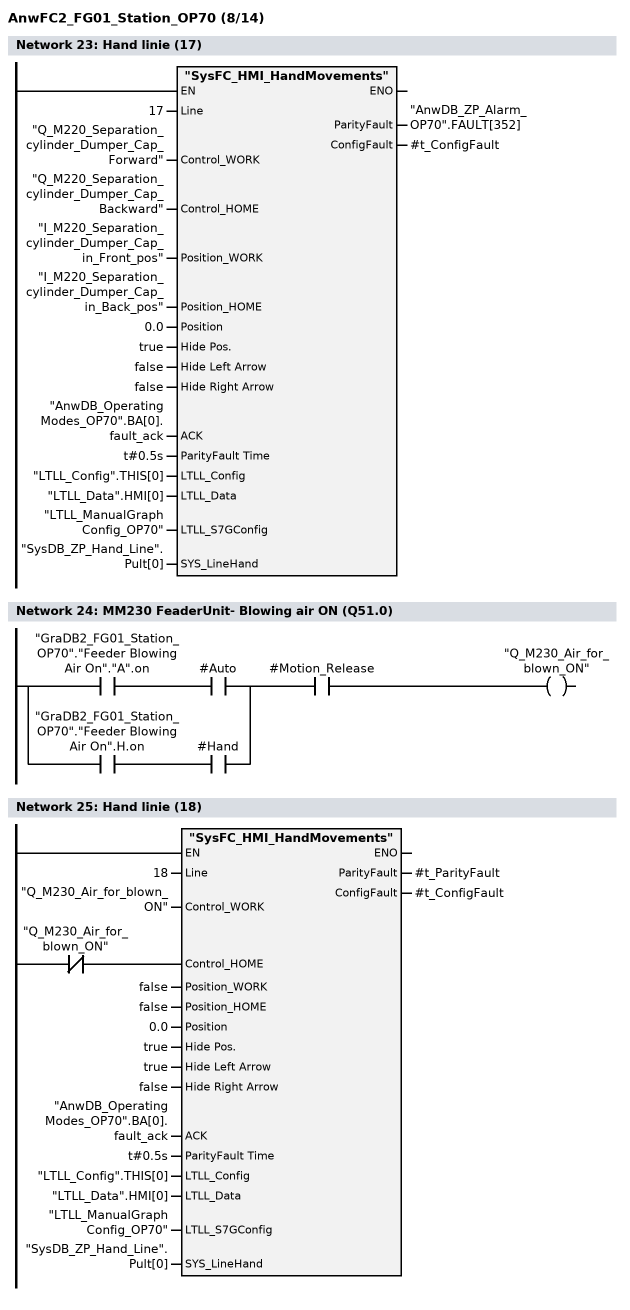
   RUNG wire#powerrail
      "SysFC_HMI_HandMovements"(Line := 17, Control_WORK := "Q_M220_Separation_cylinder_Dumper_Cap_Forward", Control_HOME := "Q_M220_Separation_cylinder_Dumper_Cap_Backward", Position_WORK := "I_M220_Separation_cylinder_Dumper_Cap_in_Front_pos", Position_HOME := "I_M220_Separation_cylinder_Dumper_Cap_in_Back_pos", Position := 0.0, "Hide Pos." := true, "Hide Left Arrow" := false, "Hide Right Arrow" := false, ACK := "AnwDB_OperatingModes_OP70".BA[0].fault_ack, "ParityFault Time" := t#0.5s, LTLL_Config := "LTLL_Config".THIS[0], LTLL_Data := "LTLL_Data".HMI[0], LTLL_S7GConfig := "LTLL_ManualGraphConfig_OP70", SYS_LineHand := "SysDB_ZP_Hand_Line".Pult[0], ParityFault => "AnwDB_ZP_Alarm_OP70".FAULT[352], ConfigFault => #t_ConfigFault)
   END_RUNG
   // the same network as SCL:
   "SysFC_HMI_HandMovements"(Line := 17,
                           Control_WORK := "Q_M220_Separation_cylinder_Dumper_Cap_Forward",
                           Control_HOME := "Q_M220_Separation_cylinder_Dumper_Cap_Backward",
                           Position_WORK := "I_M220_Separation_cylinder_Dumper_Cap_in_Front_pos",
                           Position_HOME := "I_M220_Separation_cylinder_Dumper_Cap_in_Back_pos",
                           Position := 0.0,
                           "Hide Pos." := true,
                           "Hide Left Arrow" := false,
                           "Hide Right Arrow" := false,
                           ACK := "AnwDB_OperatingModes_OP70".BA[0].fault_ack,
                           "ParityFault Time" := t#0.5s,
                           LTLL_Config := "LTLL_Config".THIS[0],
                           LTLL_Data := "LTLL_Data".HMI[0],
                           LTLL_S7GConfig := "LTLL_ManualGraphConfig_OP70",
                           SYS_LineHand := "SysDB_ZP_Hand_Line".Pult[0],
                           ParityFault => "AnwDB_ZP_Alarm_OP70".FAULT[352],
                           ConfigFault => #t_ConfigFault);
END_REGION

REGION Network 24: MM230 FeaderUnit- Blowing air ON (Q51.0)
   RUNG wire#powerrail
      Contact( "GraDB2_FG01_Station_OP70"."Feeder Blowing Air On"."A".on )
      Contact( #Auto )
      wire#w1
      Contact( #Motion_Release )
      Coil( "Q_M230_Air_for_blown_ON" )
   END_RUNG
   RUNG wire#powerrail
      Contact( "GraDB2_FG01_Station_OP70"."Feeder Blowing Air On".H.on )
      Contact( #Hand )
   END_RUNG wire#w1
   // the same network as SCL:
   "Q_M230_Air_for_blown_ON" := (("GraDB2_FG01_Station_OP70"."Feeder Blowing Air On"."A".on AND #Auto) OR ("GraDB2_FG01_Station_OP70"."Feeder Blowing Air On".H.on AND #Hand)) AND #Motion_Release;
END_REGION

REGION Network 25: Hand linie (18)
   RUNG wire#powerrail
      "SysFC_HMI_HandMovements"(Control_HOME := wire#w1, Line := 18, Control_WORK := "Q_M230_Air_for_blown_ON", Position_WORK := false, Position_HOME := false, Position := 0.0, "Hide Pos." := true, "Hide Left Arrow" := true, "Hide Right Arrow" := false, ACK := "AnwDB_OperatingModes_OP70".BA[0].fault_ack, "ParityFault Time" := t#0.5s, LTLL_Config := "LTLL_Config".THIS[0], LTLL_Data := "LTLL_Data".HMI[0], LTLL_S7GConfig := "LTLL_ManualGraphConfig_OP70", SYS_LineHand := "SysDB_ZP_Hand_Line".Pult[0], ParityFault => #t_ParityFault, ConfigFault => #t_ConfigFault)
   END_RUNG
   RUNG wire#powerrail
      I_Contact( "Q_M230_Air_for_blown_ON" )
   END_RUNG wire#w1
   // the same network as SCL:
   "SysFC_HMI_HandMovements"(Line := 18,
                           Control_WORK := "Q_M230_Air_for_blown_ON",
                           Control_HOME := NOT "Q_M230_Air_for_blown_ON",
                           Position_WORK := false,
                           Position_HOME := false,
                           Position := 0.0,
                           "Hide Pos." := true,
                           "Hide Left Arrow" := true,
                           "Hide Right Arrow" := false,
                           ACK := "AnwDB_OperatingModes_OP70".BA[0].fault_ack,
                           "ParityFault Time" := t#0.5s,
                           LTLL_Config := "LTLL_Config".THIS[0],
                           LTLL_Data := "LTLL_Data".HMI[0],
                           LTLL_S7GConfig := "LTLL_ManualGraphConfig_OP70",
                           SYS_LineHand := "SysDB_ZP_Hand_Line".Pult[0],
                           ParityFault => #t_ParityFault,
                           ConfigFault => #t_ConfigFault);
END_REGION

REGION Network 26: ################# FEEDING DEVICE #########################
END_REGION

REGION Network 27: Power ON - at Feeder Unit
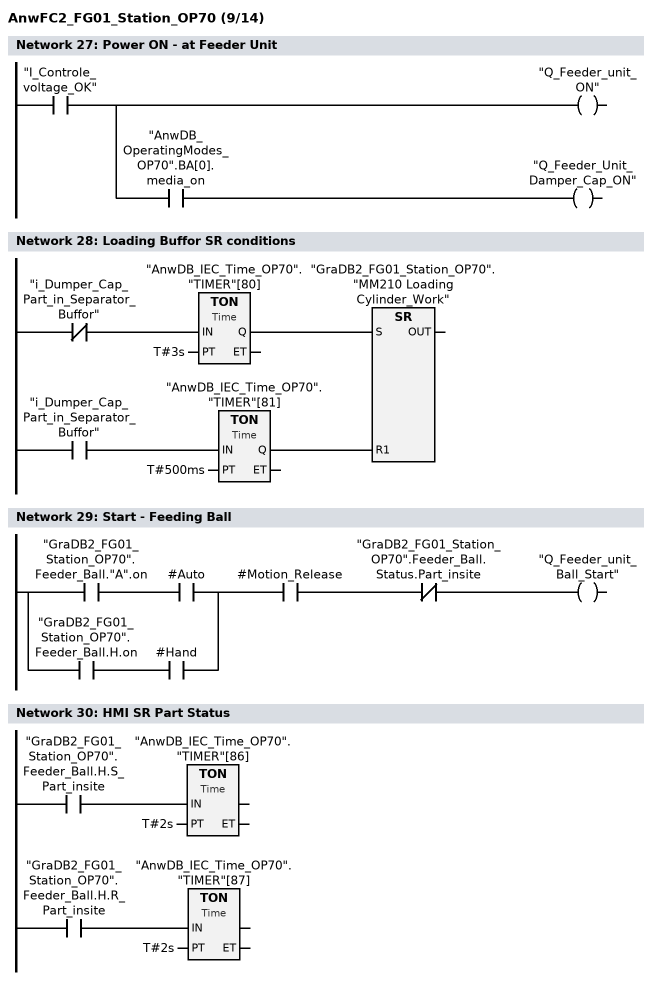
   RUNG wire#powerrail
      Contact( "I_Controle_voltage_OK" )
      wire#w1
      Coil( "Q_Feeder_unit_ON" )
   END_RUNG
   RUNG wire#w1
      Contact( "AnwDB_OperatingModes_OP70".BA[0].media_on )
      Coil( "Q_Feeder_Unit_Damper_Cap_ON" )
   END_RUNG
   // the same network as SCL:
   "Q_Feeder_unit_ON" := "I_Controle_voltage_OK";
   "Q_Feeder_Unit_Damper_Cap_ON" := "I_Controle_voltage_OK" AND "AnwDB_OperatingModes_OP70".BA[0].media_on;
END_REGION

REGION Network 28: Loading Buffor SR conditions
   RUNG wire#powerrail
      I_Contact( "i_Dumper_Cap_Part_in_Separator_Buffor" )
      { S7_Templates := "time_type := Time" } "AnwDB_IEC_Time_OP70"."TIMER"[80].TON(pt := T#3s, et =>)
      S_SR(operand := "GraDB2_FG01_Station_OP70"."MM210 Loading Cylinder_Work", r1 := wire#w1)
   END_RUNG
   RUNG wire#powerrail
      Contact( "i_Dumper_Cap_Part_in_Separator_Buffor" )
      { S7_Templates := "time_type := Time" } "AnwDB_IEC_Time_OP70"."TIMER"[81].TON(pt := T#500ms, et =>)
   END_RUNG wire#w1
   // the same network as SCL:
   "AnwDB_IEC_Time_OP70"."TIMER"[80].TON(IN := NOT "i_Dumper_Cap_Part_in_Separator_Buffor", PT := T#3s);
   #_w1 := "AnwDB_IEC_Time_OP70"."TIMER"[80].Q;
   "AnwDB_IEC_Time_OP70"."TIMER"[81].TON(IN := "i_Dumper_Cap_Part_in_Separator_Buffor", PT := T#500ms);
   IF #_w1 THEN
       "GraDB2_FG01_Station_OP70"."MM210 Loading Cylinder_Work" := TRUE;   // SR flip-flop
   END_IF;
   IF "AnwDB_IEC_Time_OP70"."TIMER"[81].Q THEN
       "GraDB2_FG01_Station_OP70"."MM210 Loading Cylinder_Work" := FALSE;
   END_IF;
END_REGION

REGION Network 29: Start - Feeding Ball
   RUNG wire#powerrail
      Contact( "GraDB2_FG01_Station_OP70".Feeder_Ball."A".on )
      Contact( #Auto )
      wire#w1
      Contact( #Motion_Release )
      I_Contact( "GraDB2_FG01_Station_OP70".Feeder_Ball.Status.Part_insite )
      Coil( "Q_Feeder_unit_Ball_Start" )
   END_RUNG
   RUNG wire#powerrail
      Contact( "GraDB2_FG01_Station_OP70".Feeder_Ball.H.on )
      Contact( #Hand )
   END_RUNG wire#w1
   // the same network as SCL:
   "Q_Feeder_unit_Ball_Start" := (("GraDB2_FG01_Station_OP70".Feeder_Ball."A".on AND #Auto) OR ("GraDB2_FG01_Station_OP70".Feeder_Ball.H.on AND #Hand)) AND #Motion_Release AND NOT "GraDB2_FG01_Station_OP70".Feeder_Ball.Status.Part_insite;
END_REGION

REGION Network 30: HMI SR Part Status
   RUNG wire#powerrail
      Contact( "GraDB2_FG01_Station_OP70".Feeder_Ball.H.S_Part_insite )
      { S7_Templates := "time_type := Time" } "AnwDB_IEC_Time_OP70"."TIMER"[86].TON(pt := T#2s, et =>)
   END_RUNG
   RUNG wire#powerrail
      Contact( "GraDB2_FG01_Station_OP70".Feeder_Ball.H.R_Part_insite )
      { S7_Templates := "time_type := Time" } "AnwDB_IEC_Time_OP70"."TIMER"[87].TON(pt := T#2s, et =>)
   END_RUNG
   // the same network as SCL:
   "AnwDB_IEC_Time_OP70"."TIMER"[86].TON(IN := "GraDB2_FG01_Station_OP70".Feeder_Ball.H.S_Part_insite,
                           PT := T#2s);
   "AnwDB_IEC_Time_OP70"."TIMER"[87].TON(IN := "GraDB2_FG01_Station_OP70".Feeder_Ball.H.R_Part_insite,
                           PT := T#2s);
END_REGION

REGION Network 31: Part Inside
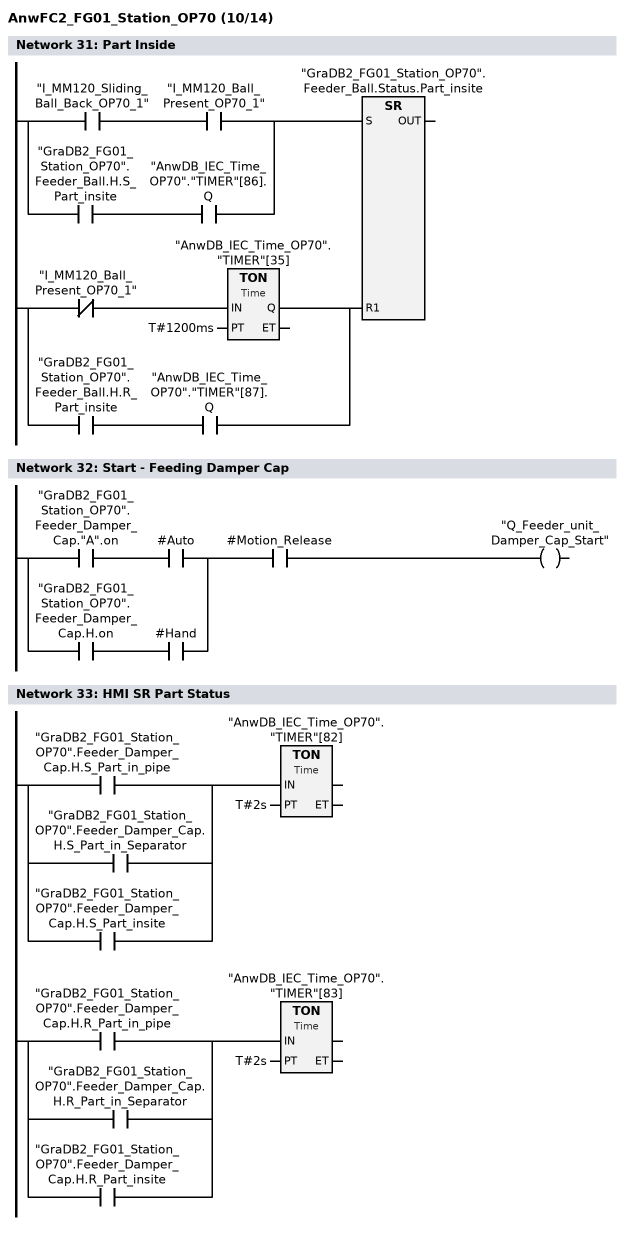
   RUNG wire#powerrail
      Contact( "I_MM120_Sliding_Ball_Back_OP70_1" )
      Contact( "I_MM120_Ball_Present_OP70_1" )
      wire#w1
      S_SR(operand := "GraDB2_FG01_Station_OP70".Feeder_Ball.Status.Part_insite, r1 := wire#w2)
   END_RUNG
   RUNG wire#powerrail
      Contact( "GraDB2_FG01_Station_OP70".Feeder_Ball.H.S_Part_insite )
      Contact( "AnwDB_IEC_Time_OP70"."TIMER"[86].Q )
   END_RUNG wire#w1
   RUNG wire#powerrail
      I_Contact( "I_MM120_Ball_Present_OP70_1" )
      { S7_Templates := "time_type := Time" } "AnwDB_IEC_Time_OP70"."TIMER"[35].TON(pt := T#1200ms, et =>)
   END_RUNG wire#w2
   RUNG wire#powerrail
      Contact( "GraDB2_FG01_Station_OP70".Feeder_Ball.H.R_Part_insite )
      Contact( "AnwDB_IEC_Time_OP70"."TIMER"[87].Q )
   END_RUNG wire#w2
   // the same network as SCL:
   #_w1 := ("I_MM120_Sliding_Ball_Back_OP70_1" AND "I_MM120_Ball_Present_OP70_1") OR ("GraDB2_FG01_Station_OP70".Feeder_Ball.H.S_Part_insite AND "AnwDB_IEC_Time_OP70"."TIMER"[86].Q);
   "AnwDB_IEC_Time_OP70"."TIMER"[35].TON(IN := NOT "I_MM120_Ball_Present_OP70_1", PT := T#1200ms);
   IF #_w1 THEN
       "GraDB2_FG01_Station_OP70".Feeder_Ball.Status.Part_insite := TRUE;   // SR flip-flop
   END_IF;
   IF "AnwDB_IEC_Time_OP70"."TIMER"[35].Q OR ("GraDB2_FG01_Station_OP70".Feeder_Ball.H.R_Part_insite AND "AnwDB_IEC_Time_OP70"."TIMER"[87].Q) THEN
       "GraDB2_FG01_Station_OP70".Feeder_Ball.Status.Part_insite := FALSE;
   END_IF;
END_REGION

REGION Network 32: Start - Feeding Damper Cap
   RUNG wire#powerrail
      Contact( "GraDB2_FG01_Station_OP70".Feeder_Damper_Cap."A".on )
      Contact( #Auto )
      wire#w1
      Contact( #Motion_Release )
      Coil( "Q_Feeder_unit_Damper_Cap_Start" )
   END_RUNG
   RUNG wire#powerrail
      Contact( "GraDB2_FG01_Station_OP70".Feeder_Damper_Cap.H.on )
      Contact( #Hand )
   END_RUNG wire#w1
   // the same network as SCL:
   "Q_Feeder_unit_Damper_Cap_Start" := (("GraDB2_FG01_Station_OP70".Feeder_Damper_Cap."A".on AND #Auto) OR ("GraDB2_FG01_Station_OP70".Feeder_Damper_Cap.H.on AND #Hand)) AND #Motion_Release;
END_REGION

REGION Network 33: HMI SR Part Status
   RUNG wire#powerrail
      Contact( "GraDB2_FG01_Station_OP70".Feeder_Damper_Cap.H.S_Part_in_pipe )
      wire#w1
      { S7_Templates := "time_type := Time" } "AnwDB_IEC_Time_OP70"."TIMER"[82].TON(pt := T#2s, et =>)
   END_RUNG
   RUNG wire#powerrail
      Contact( "GraDB2_FG01_Station_OP70".Feeder_Damper_Cap.H.S_Part_in_Separator )
   END_RUNG wire#w1
   RUNG wire#powerrail
      Contact( "GraDB2_FG01_Station_OP70".Feeder_Damper_Cap.H.S_Part_insite )
   END_RUNG wire#w1
   RUNG wire#powerrail
      Contact( "GraDB2_FG01_Station_OP70".Feeder_Damper_Cap.H.R_Part_in_pipe )
      wire#w2
      { S7_Templates := "time_type := Time" } "AnwDB_IEC_Time_OP70"."TIMER"[83].TON(pt := T#2s, et =>)
   END_RUNG
   RUNG wire#powerrail
      Contact( "GraDB2_FG01_Station_OP70".Feeder_Damper_Cap.H.R_Part_in_Separator )
   END_RUNG wire#w2
   RUNG wire#powerrail
      Contact( "GraDB2_FG01_Station_OP70".Feeder_Damper_Cap.H.R_Part_insite )
   END_RUNG wire#w2
   // the same network as SCL:
   "AnwDB_IEC_Time_OP70"."TIMER"[82].TON(IN := "GraDB2_FG01_Station_OP70".Feeder_Damper_Cap.H.S_Part_in_pipe OR "GraDB2_FG01_Station_OP70".Feeder_Damper_Cap.H.S_Part_in_Separator OR "GraDB2_FG01_Station_OP70".Feeder_Damper_Cap.H.S_Part_insite,
                           PT := T#2s);
   "AnwDB_IEC_Time_OP70"."TIMER"[83].TON(IN := "GraDB2_FG01_Station_OP70".Feeder_Damper_Cap.H.R_Part_in_pipe OR "GraDB2_FG01_Station_OP70".Feeder_Damper_Cap.H.R_Part_in_Separator OR "GraDB2_FG01_Station_OP70".Feeder_Damper_Cap.H.R_Part_insite,
                           PT := T#2s);
END_REGION

REGION Network 34: Part in Separator
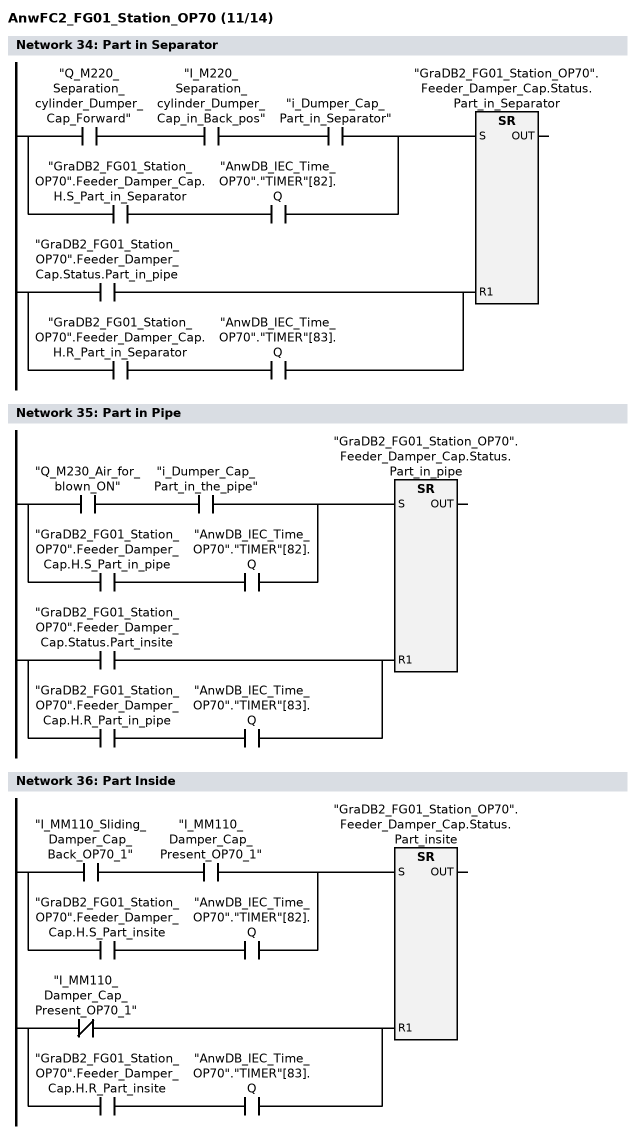
   RUNG wire#powerrail
      Contact( "Q_M220_Separation_cylinder_Dumper_Cap_Forward" )
      Contact( "I_M220_Separation_cylinder_Dumper_Cap_in_Back_pos" )
      Contact( "i_Dumper_Cap_Part_in_Separator" )
      wire#w1
      S_SR(operand := "GraDB2_FG01_Station_OP70".Feeder_Damper_Cap.Status.Part_in_Separator, r1 := wire#w2)
   END_RUNG
   RUNG wire#powerrail
      Contact( "GraDB2_FG01_Station_OP70".Feeder_Damper_Cap.H.S_Part_in_Separator )
      Contact( "AnwDB_IEC_Time_OP70"."TIMER"[82].Q )
   END_RUNG wire#w1
   RUNG wire#powerrail
      Contact( "GraDB2_FG01_Station_OP70".Feeder_Damper_Cap.Status.Part_in_pipe )
   END_RUNG wire#w2
   RUNG wire#powerrail
      Contact( "GraDB2_FG01_Station_OP70".Feeder_Damper_Cap.H.R_Part_in_Separator )
      Contact( "AnwDB_IEC_Time_OP70"."TIMER"[83].Q )
   END_RUNG wire#w2
   // the same network as SCL:
   IF ("Q_M220_Separation_cylinder_Dumper_Cap_Forward" AND "I_M220_Separation_cylinder_Dumper_Cap_in_Back_pos" AND "i_Dumper_Cap_Part_in_Separator") OR ("GraDB2_FG01_Station_OP70".Feeder_Damper_Cap.H.S_Part_in_Separator AND "AnwDB_IEC_Time_OP70"."TIMER"[82].Q) THEN
       "GraDB2_FG01_Station_OP70".Feeder_Damper_Cap.Status.Part_in_Separator := TRUE;   // SR flip-flop
   END_IF;
   IF "GraDB2_FG01_Station_OP70".Feeder_Damper_Cap.Status.Part_in_pipe OR ("GraDB2_FG01_Station_OP70".Feeder_Damper_Cap.H.R_Part_in_Separator AND "AnwDB_IEC_Time_OP70"."TIMER"[83].Q) THEN
       "GraDB2_FG01_Station_OP70".Feeder_Damper_Cap.Status.Part_in_Separator := FALSE;
   END_IF;
END_REGION

REGION Network 35: Part in Pipe
   RUNG wire#powerrail
      Contact( "Q_M230_Air_for_blown_ON" )
      Contact( "i_Dumper_Cap_Part_in_the_pipe" )
      wire#w1
      S_SR(operand := "GraDB2_FG01_Station_OP70".Feeder_Damper_Cap.Status.Part_in_pipe, r1 := wire#w2)
   END_RUNG
   RUNG wire#powerrail
      Contact( "GraDB2_FG01_Station_OP70".Feeder_Damper_Cap.H.S_Part_in_pipe )
      Contact( "AnwDB_IEC_Time_OP70"."TIMER"[82].Q )
   END_RUNG wire#w1
   RUNG wire#powerrail
      Contact( "GraDB2_FG01_Station_OP70".Feeder_Damper_Cap.Status.Part_insite )
   END_RUNG wire#w2
   RUNG wire#powerrail
      Contact( "GraDB2_FG01_Station_OP70".Feeder_Damper_Cap.H.R_Part_in_pipe )
      Contact( "AnwDB_IEC_Time_OP70"."TIMER"[83].Q )
   END_RUNG wire#w2
   // the same network as SCL:
   IF ("Q_M230_Air_for_blown_ON" AND "i_Dumper_Cap_Part_in_the_pipe") OR ("GraDB2_FG01_Station_OP70".Feeder_Damper_Cap.H.S_Part_in_pipe AND "AnwDB_IEC_Time_OP70"."TIMER"[82].Q) THEN
       "GraDB2_FG01_Station_OP70".Feeder_Damper_Cap.Status.Part_in_pipe := TRUE;   // SR flip-flop
   END_IF;
   IF "GraDB2_FG01_Station_OP70".Feeder_Damper_Cap.Status.Part_insite OR ("GraDB2_FG01_Station_OP70".Feeder_Damper_Cap.H.R_Part_in_pipe AND "AnwDB_IEC_Time_OP70"."TIMER"[83].Q) THEN
       "GraDB2_FG01_Station_OP70".Feeder_Damper_Cap.Status.Part_in_pipe := FALSE;
   END_IF;
END_REGION

REGION Network 36: Part Inside
   RUNG wire#powerrail
      Contact( "I_MM110_Sliding_Damper_Cap_Back_OP70_1" )
      Contact( "I_MM110_Damper_Cap_Present_OP70_1" )
      wire#w1
      S_SR(operand := "GraDB2_FG01_Station_OP70".Feeder_Damper_Cap.Status.Part_insite, r1 := wire#w2)
   END_RUNG
   RUNG wire#powerrail
      Contact( "GraDB2_FG01_Station_OP70".Feeder_Damper_Cap.H.S_Part_insite )
      Contact( "AnwDB_IEC_Time_OP70"."TIMER"[82].Q )
   END_RUNG wire#w1
   RUNG wire#powerrail
      I_Contact( "I_MM110_Damper_Cap_Present_OP70_1" )
   END_RUNG wire#w2
   RUNG wire#powerrail
      Contact( "GraDB2_FG01_Station_OP70".Feeder_Damper_Cap.H.R_Part_insite )
      Contact( "AnwDB_IEC_Time_OP70"."TIMER"[83].Q )
   END_RUNG wire#w2
   // the same network as SCL:
   IF ("I_MM110_Sliding_Damper_Cap_Back_OP70_1" AND "I_MM110_Damper_Cap_Present_OP70_1") OR ("GraDB2_FG01_Station_OP70".Feeder_Damper_Cap.H.S_Part_insite AND "AnwDB_IEC_Time_OP70"."TIMER"[82].Q) THEN
       "GraDB2_FG01_Station_OP70".Feeder_Damper_Cap.Status.Part_insite := TRUE;   // SR flip-flop
   END_IF;
   IF NOT "I_MM110_Damper_Cap_Present_OP70_1" OR ("GraDB2_FG01_Station_OP70".Feeder_Damper_Cap.H.R_Part_insite AND "AnwDB_IEC_Time_OP70"."TIMER"[83].Q) THEN
       "GraDB2_FG01_Station_OP70".Feeder_Damper_Cap.Status.Part_insite := FALSE;
   END_IF;
END_REGION

REGION Network 37: ################# PROCES STATUS #########################
END_REGION

REGION Network 38: BEA 1 - Ebit 1
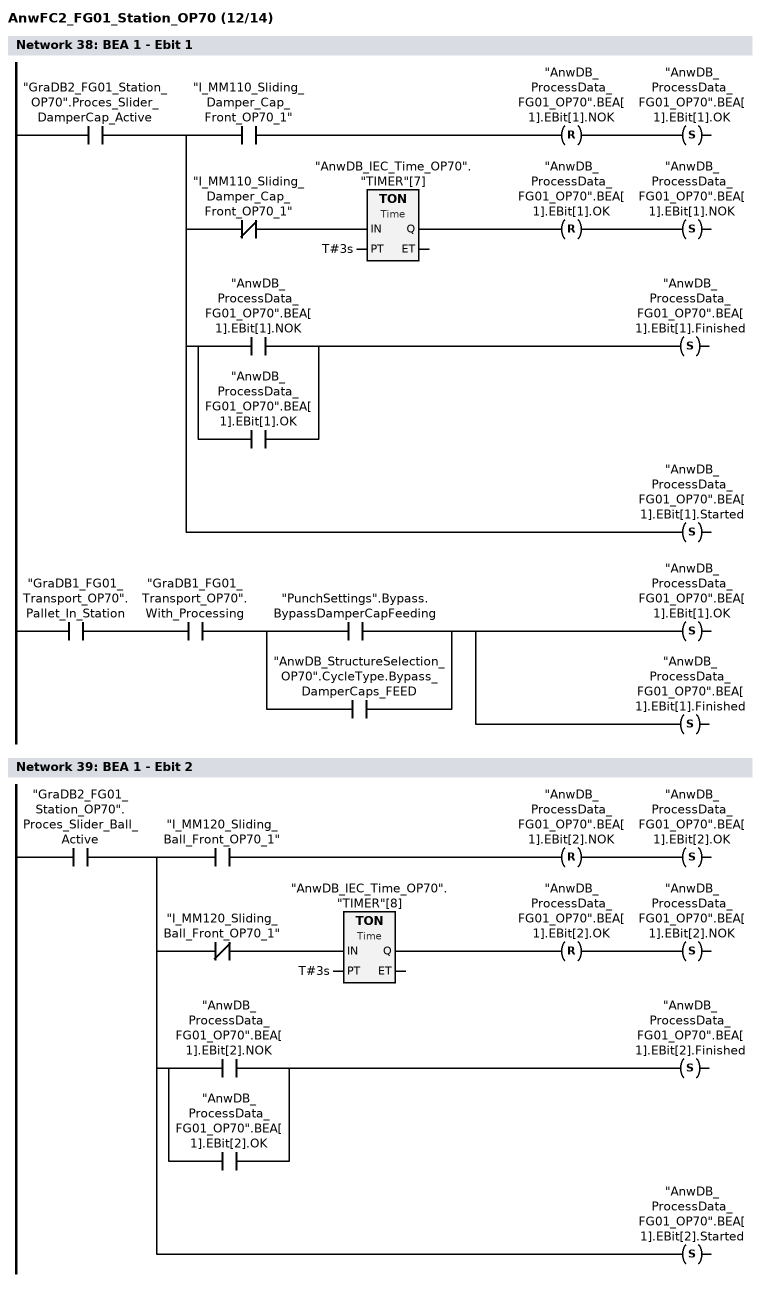
   RUNG wire#powerrail
      Contact( "GraDB2_FG01_Station_OP70".Proces_Slider_DamperCap_Active )
      wire#w1
      Contact( "I_MM110_Sliding_Damper_Cap_Front_OP70_1" )
      R_Coil( "AnwDB_ProcessData_FG01_OP70".BEA[1].EBit[1].NOK )
      S_Coil( "AnwDB_ProcessData_FG01_OP70".BEA[1].EBit[1].OK )
   END_RUNG
   RUNG wire#w1
      I_Contact( "I_MM110_Sliding_Damper_Cap_Front_OP70_1" )
      { S7_Templates := "time_type := Time" } "AnwDB_IEC_Time_OP70"."TIMER"[7].TON(pt := T#3s, et =>)
      R_Coil( "AnwDB_ProcessData_FG01_OP70".BEA[1].EBit[1].OK )
      S_Coil( "AnwDB_ProcessData_FG01_OP70".BEA[1].EBit[1].NOK )
   END_RUNG
   RUNG wire#w1
      Contact( "AnwDB_ProcessData_FG01_OP70".BEA[1].EBit[1].NOK )
      wire#w2
      S_Coil( "AnwDB_ProcessData_FG01_OP70".BEA[1].EBit[1].Finished )
   END_RUNG
   RUNG wire#w1
      Contact( "AnwDB_ProcessData_FG01_OP70".BEA[1].EBit[1].OK )
   END_RUNG wire#w2
   RUNG wire#w1
      S_Coil( "AnwDB_ProcessData_FG01_OP70".BEA[1].EBit[1].Started )
   END_RUNG
   RUNG wire#powerrail
      Contact( "GraDB1_FG01_Transport_OP70".Pallet_In_Station )
      Contact( "GraDB1_FG01_Transport_OP70".With_Processing )
      wire#w3
      Contact( "PunchSettings".Bypass.BypassDamperCapFeeding )
      wire#w4
      S_Coil( "AnwDB_ProcessData_FG01_OP70".BEA[1].EBit[1].OK )
   END_RUNG
   RUNG wire#w3
      Contact( "AnwDB_StructureSelection_OP70".CycleType.Bypass_DamperCaps_FEED )
   END_RUNG wire#w4
   RUNG wire#w4
      S_Coil( "AnwDB_ProcessData_FG01_OP70".BEA[1].EBit[1].Finished )
   END_RUNG
   // the same network as SCL:
   IF "GraDB2_FG01_Station_OP70".Proces_Slider_DamperCap_Active AND "I_MM110_Sliding_Damper_Cap_Front_OP70_1" THEN
       "AnwDB_ProcessData_FG01_OP70".BEA[1].EBit[1].NOK := FALSE;
       "AnwDB_ProcessData_FG01_OP70".BEA[1].EBit[1].OK := TRUE;
   END_IF;
   "AnwDB_IEC_Time_OP70"."TIMER"[7].TON(IN := "GraDB2_FG01_Station_OP70".Proces_Slider_DamperCap_Active AND NOT "I_MM110_Sliding_Damper_Cap_Front_OP70_1",
                           PT := T#3s);
   IF "AnwDB_IEC_Time_OP70"."TIMER"[7].Q THEN
       "AnwDB_ProcessData_FG01_OP70".BEA[1].EBit[1].OK := FALSE;
       "AnwDB_ProcessData_FG01_OP70".BEA[1].EBit[1].NOK := TRUE;
   END_IF;
   IF "GraDB2_FG01_Station_OP70".Proces_Slider_DamperCap_Active AND ("AnwDB_ProcessData_FG01_OP70".BEA[1].EBit[1].NOK OR "AnwDB_ProcessData_FG01_OP70".BEA[1].EBit[1].OK) THEN
       "AnwDB_ProcessData_FG01_OP70".BEA[1].EBit[1].Finished := TRUE;
   END_IF;
   IF "GraDB2_FG01_Station_OP70".Proces_Slider_DamperCap_Active THEN
       "AnwDB_ProcessData_FG01_OP70".BEA[1].EBit[1].Started := TRUE;
   END_IF;
   IF "GraDB1_FG01_Transport_OP70".Pallet_In_Station AND "GraDB1_FG01_Transport_OP70".With_Processing AND ("PunchSettings".Bypass.BypassDamperCapFeeding OR "AnwDB_StructureSelection_OP70".CycleType.Bypass_DamperCaps_FEED) THEN
       "AnwDB_ProcessData_FG01_OP70".BEA[1].EBit[1].OK := TRUE;
       "AnwDB_ProcessData_FG01_OP70".BEA[1].EBit[1].Finished := TRUE;
   END_IF;
END_REGION

REGION Network 39: BEA 1 - Ebit 2
   RUNG wire#powerrail
      Contact( "GraDB2_FG01_Station_OP70".Proces_Slider_Ball_Active )
      wire#w1
      Contact( "I_MM120_Sliding_Ball_Front_OP70_1" )
      R_Coil( "AnwDB_ProcessData_FG01_OP70".BEA[1].EBit[2].NOK )
      S_Coil( "AnwDB_ProcessData_FG01_OP70".BEA[1].EBit[2].OK )
   END_RUNG
   RUNG wire#w1
      I_Contact( "I_MM120_Sliding_Ball_Front_OP70_1" )
      { S7_Templates := "time_type := Time" } "AnwDB_IEC_Time_OP70"."TIMER"[8].TON(pt := T#3s, et =>)
      R_Coil( "AnwDB_ProcessData_FG01_OP70".BEA[1].EBit[2].OK )
      S_Coil( "AnwDB_ProcessData_FG01_OP70".BEA[1].EBit[2].NOK )
   END_RUNG
   RUNG wire#w1
      Contact( "AnwDB_ProcessData_FG01_OP70".BEA[1].EBit[2].NOK )
      wire#w2
      S_Coil( "AnwDB_ProcessData_FG01_OP70".BEA[1].EBit[2].Finished )
   END_RUNG
   RUNG wire#w1
      Contact( "AnwDB_ProcessData_FG01_OP70".BEA[1].EBit[2].OK )
   END_RUNG wire#w2
   RUNG wire#w1
      S_Coil( "AnwDB_ProcessData_FG01_OP70".BEA[1].EBit[2].Started )
   END_RUNG
   // the same network as SCL:
   IF "GraDB2_FG01_Station_OP70".Proces_Slider_Ball_Active AND "I_MM120_Sliding_Ball_Front_OP70_1" THEN
       "AnwDB_ProcessData_FG01_OP70".BEA[1].EBit[2].NOK := FALSE;
       "AnwDB_ProcessData_FG01_OP70".BEA[1].EBit[2].OK := TRUE;
   END_IF;
   "AnwDB_IEC_Time_OP70"."TIMER"[8].TON(IN := "GraDB2_FG01_Station_OP70".Proces_Slider_Ball_Active AND NOT "I_MM120_Sliding_Ball_Front_OP70_1",
                           PT := T#3s);
   IF "AnwDB_IEC_Time_OP70"."TIMER"[8].Q THEN
       "AnwDB_ProcessData_FG01_OP70".BEA[1].EBit[2].OK := FALSE;
       "AnwDB_ProcessData_FG01_OP70".BEA[1].EBit[2].NOK := TRUE;
   END_IF;
   IF "GraDB2_FG01_Station_OP70".Proces_Slider_Ball_Active AND ("AnwDB_ProcessData_FG01_OP70".BEA[1].EBit[2].NOK OR "AnwDB_ProcessData_FG01_OP70".BEA[1].EBit[2].OK) THEN
       "AnwDB_ProcessData_FG01_OP70".BEA[1].EBit[2].Finished := TRUE;
   END_IF;
   IF "GraDB2_FG01_Station_OP70".Proces_Slider_Ball_Active THEN
       "AnwDB_ProcessData_FG01_OP70".BEA[1].EBit[2].Started := TRUE;
   END_IF;
END_REGION

REGION Network 40: BEA 2 Ebit 1
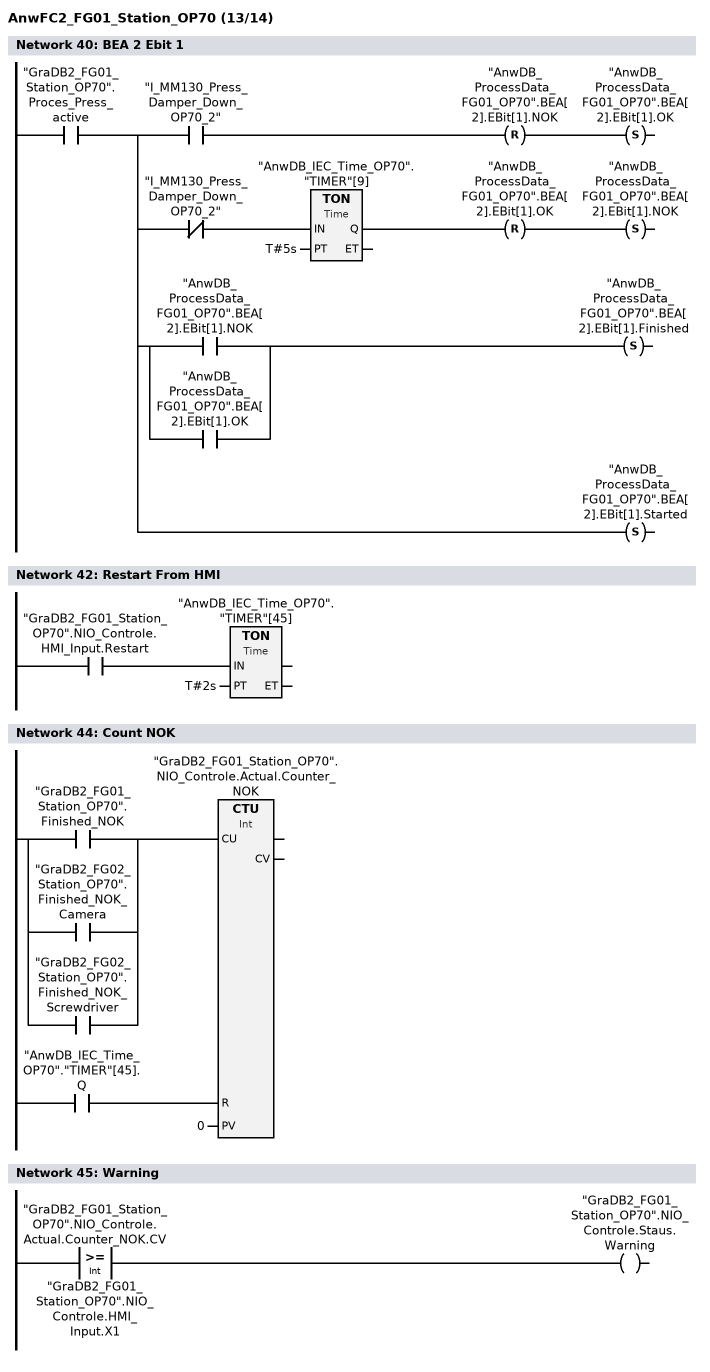
   RUNG wire#powerrail
      Contact( "GraDB2_FG01_Station_OP70".Proces_Press_active )
      wire#w1
      Contact( "I_MM130_Press_Damper_Down_OP70_2" )
      R_Coil( "AnwDB_ProcessData_FG01_OP70".BEA[2].EBit[1].NOK )
      S_Coil( "AnwDB_ProcessData_FG01_OP70".BEA[2].EBit[1].OK )
   END_RUNG
   RUNG wire#w1
      I_Contact( "I_MM130_Press_Damper_Down_OP70_2" )
      { S7_Templates := "time_type := Time" } "AnwDB_IEC_Time_OP70"."TIMER"[9].TON(pt := T#5s, et =>)
      R_Coil( "AnwDB_ProcessData_FG01_OP70".BEA[2].EBit[1].OK )
      S_Coil( "AnwDB_ProcessData_FG01_OP70".BEA[2].EBit[1].NOK )
   END_RUNG
   RUNG wire#w1
      Contact( "AnwDB_ProcessData_FG01_OP70".BEA[2].EBit[1].NOK )
      wire#w2
      S_Coil( "AnwDB_ProcessData_FG01_OP70".BEA[2].EBit[1].Finished )
   END_RUNG
   RUNG wire#w1
      Contact( "AnwDB_ProcessData_FG01_OP70".BEA[2].EBit[1].OK )
   END_RUNG wire#w2
   RUNG wire#w1
      S_Coil( "AnwDB_ProcessData_FG01_OP70".BEA[2].EBit[1].Started )
   END_RUNG
   // the same network as SCL:
   IF "GraDB2_FG01_Station_OP70".Proces_Press_active AND "I_MM130_Press_Damper_Down_OP70_2" THEN
       "AnwDB_ProcessData_FG01_OP70".BEA[2].EBit[1].NOK := FALSE;
       "AnwDB_ProcessData_FG01_OP70".BEA[2].EBit[1].OK := TRUE;
   END_IF;
   "AnwDB_IEC_Time_OP70"."TIMER"[9].TON(IN := "GraDB2_FG01_Station_OP70".Proces_Press_active AND NOT "I_MM130_Press_Damper_Down_OP70_2",
                           PT := T#5s);
   IF "AnwDB_IEC_Time_OP70"."TIMER"[9].Q THEN
       "AnwDB_ProcessData_FG01_OP70".BEA[2].EBit[1].OK := FALSE;
       "AnwDB_ProcessData_FG01_OP70".BEA[2].EBit[1].NOK := TRUE;
   END_IF;
   IF "GraDB2_FG01_Station_OP70".Proces_Press_active AND ("AnwDB_ProcessData_FG01_OP70".BEA[2].EBit[1].NOK OR "AnwDB_ProcessData_FG01_OP70".BEA[2].EBit[1].OK) THEN
       "AnwDB_ProcessData_FG01_OP70".BEA[2].EBit[1].Finished := TRUE;
   END_IF;
   IF "GraDB2_FG01_Station_OP70".Proces_Press_active THEN
       "AnwDB_ProcessData_FG01_OP70".BEA[2].EBit[1].Started := TRUE;
   END_IF;
END_REGION

REGION Network 41: ################ NIO Counting ################
END_REGION

REGION Network 42: Restart From HMI
   RUNG wire#powerrail
      Contact( "GraDB2_FG01_Station_OP70".NIO_Controle.HMI_Input.Restart )
      { S7_Templates := "time_type := Time" } "AnwDB_IEC_Time_OP70"."TIMER"[45].TON(pt := T#2s, et =>)
   END_RUNG
   // the same network as SCL:
   "AnwDB_IEC_Time_OP70"."TIMER"[45].TON(IN := "GraDB2_FG01_Station_OP70".NIO_Controle.HMI_Input.Restart,
                           PT := T#2s);
END_REGION

REGION Network 43 (SCL): Rewrite Data from HMI
   #X1 := "GraDB2_FG01_Station_OP70".NIO_Controle.HMI_Input.X1;
   #X2 := "GraDB2_FG01_Station_OP70".NIO_Controle.HMI_Input.X2;


   REGION // Controle Input Data
       IF #X1 > #X2 THEN
           #X1 := "GraDB2_FG01_Station_OP70".NIO_Controle.HMI_Input.X1 := #X2;
       END_IF;
       IF #X1 <= 0 THEN
           #X1 := "GraDB2_FG01_Station_OP70".NIO_Controle.HMI_Input.X1 := 1;
       END_IF;

       IF #X2 <= 0 THEN
           #X2 := "GraDB2_FG01_Station_OP70".NIO_Controle.HMI_Input.X2 := 1;
       END_IF;
   END_REGION
END_REGION

REGION Network 44: Count NOK
   RUNG wire#powerrail
      Contact( "GraDB2_FG01_Station_OP70".Finished_NOK )
      wire#w1
      { S7_Templates := "value_type := Int" } "GraDB2_FG01_Station_OP70".NIO_Controle.Actual.Counter_NOK.CTU(r := wire#w2, pv := 0, cv =>)
   END_RUNG
   RUNG wire#powerrail
      Contact( "GraDB2_FG02_Station_OP70".Finished_NOK_Camera )
   END_RUNG wire#w1
   RUNG wire#powerrail
      Contact( "GraDB2_FG02_Station_OP70".Finished_NOK_Screwdriver )
   END_RUNG wire#w1
   RUNG wire#powerrail
      Contact( "AnwDB_IEC_Time_OP70"."TIMER"[45].Q )
   END_RUNG wire#w2
   // the same network as SCL:
   "GraDB2_FG01_Station_OP70".NIO_Controle.Actual.Counter_NOK.CTU(CU := "GraDB2_FG01_Station_OP70".Finished_NOK OR "GraDB2_FG02_Station_OP70".Finished_NOK_Camera OR "GraDB2_FG02_Station_OP70".Finished_NOK_Screwdriver,
                           R := "AnwDB_IEC_Time_OP70"."TIMER"[45].Q,
                           PV := 0);
END_REGION

REGION Network 45: Warning
   RUNG wire#powerrail
      { S7_Templates := "SrcType := Int" } GE_Contact(in1 := "GraDB2_FG01_Station_OP70".NIO_Controle.Actual.Counter_NOK.CV, in2 := "GraDB2_FG01_Station_OP70".NIO_Controle.HMI_Input.X1)
      Coil( "GraDB2_FG01_Station_OP70".NIO_Controle.Staus.Warning )
   END_RUNG
   // the same network as SCL:
   "GraDB2_FG01_Station_OP70".NIO_Controle.Staus.Warning := "GraDB2_FG01_Station_OP70".NIO_Controle.Actual.Counter_NOK.CV >= "GraDB2_FG01_Station_OP70".NIO_Controle.HMI_Input.X1;
END_REGION

REGION Network 46: Error
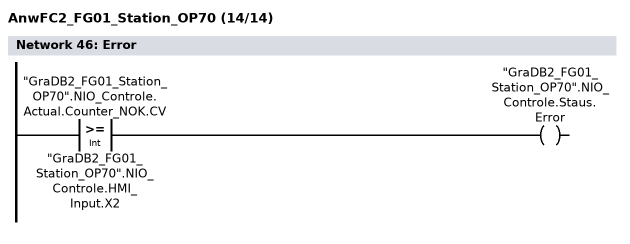
   RUNG wire#powerrail
      { S7_Templates := "SrcType := Int" } GE_Contact(in1 := "GraDB2_FG01_Station_OP70".NIO_Controle.Actual.Counter_NOK.CV, in2 := "GraDB2_FG01_Station_OP70".NIO_Controle.HMI_Input.X2)
      Coil( "GraDB2_FG01_Station_OP70".NIO_Controle.Staus.Error )
   END_RUNG
   // the same network as SCL:
   "GraDB2_FG01_Station_OP70".NIO_Controle.Staus.Error := "GraDB2_FG01_Station_OP70".NIO_Controle.Actual.Counter_NOK.CV >= "GraDB2_FG01_Station_OP70".NIO_Controle.HMI_Input.X2;
END_REGION
END_FUNCTION
